LIN {X 0,Y 172.638,Z 369.1,A -85,B 0,C 180,E1 -26067.806,E2 -26067.806} C_VEL
LIN {X 0,Y 170.453,Z 370.698,A -85,B 0,C 180,E1 -26067.724,E2 -26067.724} C_VEL
LIN {X 0,Y 167.759,Z 372.433,A -85,B 0,C 180,E1 -26068.163,E2 -26068.163} C_VEL
LIN {X 0,Y 165.128,Z 374.03,A -85,B 0,C 180,E1 -26069.021,E2 -26069.021} C_VEL
LIN {X 0,Y 159.69,Z 377.088,A -85,B 0,C 180,E1 -26071.335,E2 -26071.335} C_VEL
LIN {X 0,Y 157.543,Z 378.251,A -85,B 0,C 180,E1 -26071.948,E2 -26071.948} C_VEL
LIN {X 0,Y 147.13,Z 383.164,A -85,B 0,C 180,E1 -26074.539,E2 -26074.539} C_VEL
LIN {X 0,Y 136.791,Z 386.889,A -85,B 0,C 180,E1 -26077.644,E2 -26077.644} C_VEL
LIN {X 0,Y 125.587,Z 389.614,A -85,B 0,C 180,E1 -26082.061,E2 -26082.061} C_VEL
LIN {X 0,Y 115.177,Z 390.768,A -85,B 0,C 180,E1 -26087.515,E2 -26087.515} C_VEL
LIN {X 0,Y 105.941,Z 390.198,A -85,B 0,C 180,E1 -26094.344,E2 -26094.344} C_VEL
LIN {X 0,Y 100.509,Z 388.699,A -85,B 0,C 180,E1 -26100.001,E2 -26100.001} C_VEL
LIN {X 0,Y 97.504,Z 387.177,A -85,B 0,C 180,E1 -26104.134,E2 -26104.134} C_VEL
LIN {X 0,Y 93.505,Z 383.221,A -85,B 0,C 180,E1 -26112.269,E2 -26112.269} C_VEL
LIN {X 0,Y 91.521,Z 378.192,A -85,B 0,C 180,E1 -26120.181,E2 -26120.181} C_VEL
LIN {X 0,Y 91.194,Z 372.228,A -85,B 0,C 180,E1 -26127.543,E2 -26127.543} C_VEL
LIN {X 0,Y 91.607,Z 365.87,A -85,B 0,C 180,E1 -26133.796,E2 -26133.796} C_VEL
LIN {X 0,Y 92.588,Z 357.724,A -85,B 0,C 180,E1 -26140.216,E2 -26140.216} C_VEL
LIN {X 0,Y 94.126,Z 348.531,A -85,B 0,C 180,E1 -26145.946,E2 -26145.946} C_VEL
LIN {X 0,Y 96.068,Z 338.761,A -85,B 0,C 180,E1 -26150.765,E2 -26150.765} C_VEL
LIN {X 0,Y 98.32,Z 327.543,A -85,B 0,C 180,E1 -26155.117,E2 -26155.117} C_VEL
LIN {X 0,Y 100.753,Z 315.315,A -85,B 0,C 180,E1 -26158.707,E2 -26158.707} C_VEL
LIN {X 0,Y 102.943,Z 302.841,A -85,B 0,C 180,E1 -26161.448,E2 -26161.448} C_VEL
LIN {X 0,Y 104.614,Z 289.402,A -85,B 0,C 180,E1 -26163.561,E2 -26163.561} C_VEL
LIN {X 0,Y 106.685,Z 268.345,A -85,B 0,C 180,E1 -26165.639,E2 -26165.639} C_VEL
LIN {X 0,Y 109.722,Z 233.038,A -85,B 0,C 180,E1 -26168.778,E2 -26168.778} C_VEL
LIN {X 0,Y 103.431,Z 215.21,A -85,B 0,C 180,E1 -26172.045,E2 -26172.045} C_VEL
LIN {X 0,Y 97.31,Z 199.967,A -85,B 0,C 180,E1 -26175.421,E2 -26175.421} C_VEL
LIN {X 0,Y 94.113,Z 192.132,A -85,B 0,C 180,E1 -26177.325,E2 -26177.325} C_VEL
LIN {X 0,Y 94.078,Z 191.767,A -85,B 0,C 180,E1 -26177.594,E2 -26177.594} C_VEL
LIN {X 0,Y 94.163,Z 191.756,A -85,B 0,C 180,E1 -26181.411,E2 -26181.411} C_VEL
LIN {X 0,Y 94.758,Z 191.674,A -85,B 0,C 180,E1 -26189.996,E2 -26189.996} C_VEL
LIN {X 0,Y 94.134,Z 191.751,A -85,B 0,C 180,E1 -26198.584,E2 -26198.584} C_VEL
LIN {X 0,Y 93.959,Z 191.781,A -85,B 0,C 180,E1 -26203.492,E2 -26203.492} C_VEL
LIN {X 0,Y 93.642,Z 191.82,A -85,B 0,C 180,E1 -26212.036,E2 -26212.036} C_VEL
LIN {X 0,Y 93.586,Z 191.823,A -85,B 0,C 180,E1 -26216.777,E2 -26216.777} C_VEL
LIN {X 0,Y 93.58,Z 191.822,A -85,B 0,C 180,E1 -26224.296,E2 -26224.296} C_VEL
LIN {X 0,Y 93.524,Z 191.827,A -85,B 0,C 180,E1 -26232.551,E2 -26232.551} C_VEL
LIN {X 0,Y 93.527,Z 191.83,A -85,B 0,C 180,E1 -26238.71,E2 -26238.71} C_VEL
LIN {X 0,Y 93.579,Z 191.827,A -85,B 0,C 180,E1 -26245.695,E2 -26245.695} C_VEL
LIN {X 0,Y 93.637,Z 191.82,A -85,B 0,C 180,E1 -26254.237,E2 -26254.237} C_VEL
LIN {X 0,Y 93.646,Z 191.813,A -85,B 0,C 180,E1 -26257.96,E2 -26257.96} C_VEL
LIN {X 0,Y 94.009,Z 191.771,A -85,B 0,C 180,E1 -26267.039,E2 -26267.039} C_VEL
LIN {X 0,Y 94.152,Z 191.756,A -85,B 0,C 180,E1 -26271.413,E2 -26271.413} C_VEL
LIN {X 0,Y 94.749,Z 191.68,A -85,B 0,C 180,E1 -26279.999,E2 -26279.999} C_VEL
LIN {X 0,Y 94.125,Z 191.758,A -85,B 0,C 180,E1 -26288.587,E2 -26288.587} C_VEL
LIN {X 0,Y 93.951,Z 191.781,A -85,B 0,C 180,E1 -26293.494,E2 -26293.494} C_VEL
LIN {X 0,Y 93.636,Z 191.821,A -85,B 0,C 180,E1 -26302.041,E2 -26302.041} C_VEL
LIN {X 0,Y 93.58,Z 191.822,A -85,B 0,C 180,E1 -26306.782,E2 -26306.782} C_VEL
LIN {X 0,Y 93.576,Z 191.825,A -85,B 0,C 180,E1 -26314.301,E2 -26314.301} C_VEL
LIN {X 0,Y 93.585,Z 191.828,A -85,B 0,C 180,E1 -26319.821,E2 -26319.821} C_VEL
LIN {X 0,Y 94.705,Z 194.871,A -85,B 0,C 180,E1 -26320.588,E2 -26320.588} C_VEL
LIN {X 0,Y 101.84,Z 211.018,A -85,B 0,C 180,E1 -26324.497,E2 -26324.497} C_VEL
LIN {X 0,Y 108.216,Z 233.918,A -85,B 0,C 180,E1 -26328.406,E2 -26328.406} C_VEL
LIN {X 0,Y 108.775,Z 238.103,A -85,B 0,C 180,E1 -26328.95,E2 -26328.95} C_VEL
LIN {X 0,Y 109.169,Z 245.942,A -85,B 0,C 180,E1 -26329.835,E2 -26329.835} C_VEL
LIN {X 0,Y 105.151,Z 291.907,A -85,B 0,C 180,E1 -26334.066,E2 -26334.066} C_VEL
LIN {X 0,Y 103.46,Z 304.913,A -85,B 0,C 180,E1 -26335.92,E2 -26335.92} C_VEL
LIN {X 0,Y 101.232,Z 318.223,A -85,B 0,C 180,E1 -26338.626,E2 -26338.626} C_VEL
LIN {X 0,Y 98.938,Z 330.029,A -85,B 0,C 180,E1 -26341.931,E2 -26341.931} C_VEL
LIN {X 0,Y 96.46,Z 342.113,A -85,B 0,C 180,E1 -26346.38,E2 -26346.38} C_VEL
LIN {X 0,Y 94.41,Z 352.803,A -85,B 0,C 180,E1 -26351.56,E2 -26351.56} C_VEL
LIN {X 0,Y 93.041,Z 361.54,A -85,B 0,C 180,E1 -26356.906,E2 -26356.906} C_VEL
LIN {X 0,Y 92.355,Z 368.876,A -85,B 0,C 180,E1 -26362.495,E2 -26362.495} C_VEL
LIN {X 0,Y 92.285,Z 375.689,A -85,B 0,C 180,E1 -26368.913,E2 -26368.913} C_VEL
LIN {X 0,Y 92.355,Z 378.572,A -85,B 0,C 180,E1 -26372.184,E2 -26372.184} C_VEL
LIN {X 0,Y 92.189,Z 383.199,A -85,B 0,C 180,E1 -26378.774,E2 -26378.774} C_VEL
LIN {X 0,Y 93.115,Z 386.821,A -85,B 0,C 180,E1 -26385.321,E2 -26385.321} C_VEL
LIN {X 0,Y 95.224,Z 389.563,A -85,B 0,C 180,E1 -26391.659,E2 -26391.659} C_VEL
LIN {X 0,Y 99.89,Z 392.01,A -85,B 0,C 180,E1 -26399.509,E2 -26399.509} C_VEL
LIN {X 0,Y 106.598,Z 393.144,A -85,B 0,C 180,E1 -26406.4,E2 -26406.4} C_VEL
LIN {X 0,Y 114.858,Z 392.97,A -85,B 0,C 180,E1 -26412.309,E2 -26412.309} C_VEL
LIN {X 0,Y 124.234,Z 391.453,A -85,B 0,C 180,E1 -26417.346,E2 -26417.346} C_VEL
LIN {X 0,Y 134.749,Z 388.583,A -85,B 0,C 180,E1 -26421.479,E2 -26421.479} C_VEL
LIN {X 0,Y 146.079,Z 384.264,A -85,B 0,C 180,E1 -26424.878,E2 -26424.878} C_VEL
LIN {X 0,Y 154.429,Z 380.236,A -85,B 0,C 180,E1 -26426.9,E2 -26426.9} C_VEL
LIN {X 0,Y 164.165,Z 374.602,A -85,B 0,C 180,E1 -26428.898,E2 -26428.898} C_VEL
LIN {X 0,Y 166.024,Z 373.418,A -85,B 0,C 180,E1 -26429.237,E2 -26429.237} C_VEL
LIN {X 0,Y 167.851,Z 372.157,A -85,B 0,C 180,E1 -26429.839,E2 -26429.839} C_VEL
LIN {X 0,Y 157.543,Z 378.251,A -85,B 0,C 180,E1 -26431.948,E2 -26431.948} C_VEL
LIN {X 0,Y 152.658,Z 380.71,A -85,B 0,C 180,E1 -26432.791,E2 -26432.791} C_VEL
LIN {X 0,Y 140.141,Z 385.717,A -85,B 0,C 180,E1 -26434.113,E2 -26434.113} C_VEL
LIN {X 0,Y 134.791,Z 387.382,A -85,B 0,C 180,E1 -26434.902,E2 -26434.902} C_VEL
LIN {X 0,Y 129.86,Z 388.621,A -85,B 0,C 180,E1 -26436.166,E2 -26436.166} C_VEL
LIN {X 0,Y 119.503,Z 390.467,A -85,B 0,C 180,E1 -26440.222,E2 -26440.222} C_VEL
LIN {X 0,Y 108.749,Z 391.045,A -85,B 0,C 180,E1 -26445.799,E2 -26445.799} C_VEL
LIN {X 0,Y 100.286,Z 390.123,A -85,B 0,C 180,E1 -26451.944,E2 -26451.944} C_VEL
LIN {X 0,Y 92.745,Z 387.564,A -85,B 0,C 180,E1 -26460.001,E2 -26460.001} C_VEL
LIN {X 0,Y 88.53,Z 384.524,A -85,B 0,C 180,E1 -26466.84,E2 -26466.84} C_VEL
LIN {X 0,Y 85.732,Z 380.425,A -85,B 0,C 180,E1 -26474.238,E2 -26474.238} C_VEL
LIN {X 0,Y 84.452,Z 375.617,A -85,B 0,C 180,E1 -26481.4,E2 -26481.4} C_VEL
LIN {X 0,Y 84.254,Z 369.652,A -85,B 0,C 180,E1 -26488.663,E2 -26488.663} C_VEL
LIN {X 0,Y 84.83,Z 362.659,A -85,B 0,C 180,E1 -26495.448,E2 -26495.448} C_VEL
LIN {X 0,Y 86.008,Z 353.907,A -85,B 0,C 180,E1 -26502.219,E2 -26502.219} C_VEL
LIN {X 0,Y 87.916,Z 343.463,A -85,B 0,C 180,E1 -26508.52,E2 -26508.52} C_VEL
LIN {X 0,Y 89.928,Z 333.534,A -85,B 0,C 180,E1 -26513.232,E2 -26513.232} C_VEL
LIN {X 0,Y 92.4,Z 322.052,A -85,B 0,C 180,E1 -26517.472,E2 -26517.472} C_VEL
LIN {X 0,Y 94.926,Z 309.313,A -85,B 0,C 180,E1 -26520.983,E2 -26520.983} C_VEL
LIN {X 0,Y 96.998,Z 296.051,A -85,B 0,C 180,E1 -26523.619,E2 -26523.619} C_VEL
LIN {X 0,Y 98.656,Z 281.536,A -85,B 0,C 180,E1 -26525.543,E2 -26525.543} C_VEL
LIN {X 0,Y 103.049,Z 234.956,A -85,B 0,C 180,E1 -26529.929,E2 -26529.929} C_VEL
LIN {X 0,Y 98.97,Z 222.631,A -85,B 0,C 180,E1 -26532.297,E2 -26532.297} C_VEL
LIN {X 0,Y 92.348,Z 205.494,A -85,B 0,C 180,E1 -26536.157,E2 -26536.157} C_VEL
LIN {X 0,Y 87.771,Z 195.022,A -85,B 0,C 180,E1 -26539.047,E2 -26539.047} C_VEL
LIN {X 0,Y 87.046,Z 192.643,A -85,B 0,C 180,E1 -26539.83,E2 -26539.83} C_VEL
LIN {X 0,Y 87.688,Z 192.555,A -85,B 0,C 180,E1 -26549.996,E2 -26549.996} C_VEL
LIN {X 0,Y 87.027,Z 192.638,A -85,B 0,C 180,E1 -26559.291,E2 -26559.291} C_VEL
LIN {X 0,Y 86.86,Z 192.664,A -85,B 0,C 180,E1 -26564.044,E2 -26564.044} C_VEL
LIN {X 0,Y 86.593,Z 192.696,A -85,B 0,C 180,E1 -26568.94,E2 -26568.94} C_VEL
LIN {X 0,Y 86.554,Z 192.699,A -85,B 0,C 180,E1 -26576.722,E2 -26576.722} C_VEL
LIN {X 0,Y 86.499,Z 192.708,A -85,B 0,C 180,E1 -26585.657,E2 -26585.657} C_VEL
LIN {X 0,Y 86.468,Z 192.707,A -85,B 0,C 180,E1 -26592.985,E2 -26592.985} C_VEL
LIN {X 0,Y 86.449,Z 192.71,A -85,B 0,C 180,E1 -26599.429,E2 -26599.429} C_VEL
LIN {X 0,Y 86.523,Z 192.707,A -85,B 0,C 180,E1 -26605.346,E2 -26605.346} C_VEL
LIN {X 0,Y 86.559,Z 192.703,A -85,B 0,C 180,E1 -26613.259,E2 -26613.259} C_VEL
LIN {X 0,Y 86.592,Z 192.699,A -85,B 0,C 180,E1 -26621.054,E2 -26621.054} C_VEL
LIN {X 0,Y 86.856,Z 192.658,A -85,B 0,C 180,E1 -26626.148,E2 -26626.148} C_VEL
LIN {X 0,Y 87.055,Z 192.64,A -85,B 0,C 180,E1 -26630.707,E2 -26630.707} C_VEL
LIN {X 0,Y 87.678,Z 192.561,A -85,B 0,C 180,E1 -26639.999,E2 -26639.999} C_VEL
LIN {X 0,Y 87.019,Z 192.64,A -85,B 0,C 180,E1 -26649.295,E2 -26649.295} C_VEL
LIN {X 0,Y 86.853,Z 192.667,A -85,B 0,C 180,E1 -26654.048,E2 -26654.048} C_VEL
LIN {X 0,Y 86.585,Z 192.692,A -85,B 0,C 180,E1 -26658.945,E2 -26658.945} C_VEL
LIN {X 0,Y 86.548,Z 192.697,A -85,B 0,C 180,E1 -26666.727,E2 -26666.727} C_VEL
LIN {X 0,Y 86.471,Z 192.704,A -85,B 0,C 180,E1 -26675.641,E2 -26675.641} C_VEL
LIN {X 0,Y 86.51,Z 192.893,A -85,B 0,C 180,E1 -26677.575,E2 -26677.575} C_VEL
LIN {X 0,Y 87.529,Z 195.553,A -85,B 0,C 180,E1 -26678.319,E2 -26678.319} C_VEL
LIN {X 0,Y 92.221,Z 205.62,A -85,B 0,C 180,E1 -26681.194,E2 -26681.194} C_VEL
LIN {X 0,Y 96.159,Z 215.384,A -85,B 0,C 180,E1 -26683.52,E2 -26683.52} C_VEL
LIN {X 0,Y 102.028,Z 237.053,A -85,B 0,C 180,E1 -26687.476,E2 -26687.476} C_VEL
LIN {X 0,Y 102.435,Z 246.588,A -85,B 0,C 180,E1 -26688.628,E2 -26688.628} C_VEL
LIN {X 0,Y 98.298,Z 291.946,A -85,B 0,C 180,E1 -26693.062,E2 -26693.062} C_VEL
LIN {X 0,Y 96.341,Z 306.14,A -85,B 0,C 180,E1 -26695.26,E2 -26695.26} C_VEL
LIN {X 0,Y 94.222,Z 318.099,A -85,B 0,C 180,E1 -26697.901,E2 -26697.901} C_VEL
LIN {X 0,Y 91.871,Z 329.891,A -85,B 0,C 180,E1 -26701.442,E2 -26701.442} C_VEL
LIN {X 0,Y 89.325,Z 341.868,A -85,B 0,C 180,E1 -26706.224,E2 -26706.224} C_VEL
LIN {X 0,Y 87.44,Z 351.526,A -85,B 0,C 180,E1 -26711.25,E2 -26711.25} C_VEL
LIN {X 0,Y 86.054,Z 360.36,A -85,B 0,C 180,E1 -26717.027,E2 -26717.027} C_VEL
LIN {X 0,Y 85.397,Z 367.554,A -85,B 0,C 180,E1 -26722.814,E2 -26722.814} C_VEL
LIN {X 0,Y 85.354,Z 373.709,A -85,B 0,C 180,E1 -26728.825,E2 -26728.825} C_VEL
LIN {X 0,Y 85.445,Z 376.765,A -85,B 0,C 180,E1 -26732.361,E2 -26732.361} C_VEL
LIN {X 0,Y 85.35,Z 381.668,A -85,B 0,C 180,E1 -26739.483,E2 -26739.483} C_VEL
LIN {X 0,Y 87.053,Z 386.605,A -85,B 0,C 180,E1 -26748.844,E2 -26748.844} C_VEL
LIN {X 0,Y 90.932,Z 390.065,A -85,B 0,C 180,E1 -26757.632,E2 -26757.632} C_VEL
LIN {X 0,Y 97.206,Z 392.165,A -85,B 0,C 180,E1 -26765.342,E2 -26765.342} C_VEL
LIN {X 0,Y 105.243,Z 392.954,A -85,B 0,C 180,E1 -26771.901,E2 -26771.901} C_VEL
LIN {X 0,Y 114.484,Z 392.455,A -85,B 0,C 180,E1 -26777.452,E2 -26777.452} C_VEL
LIN {X 0,Y 124.898,Z 390.666,A -85,B 0,C 180,E1 -26781.983,E2 -26781.983} C_VEL
LIN {X 0,Y 136.239,Z 387.523,A -85,B 0,C 180,E1 -26785.631,E2 -26785.631} C_VEL
LIN {X 0,Y 148.218,Z 382.837,A -85,B 0,C 180,E1 -26788.598,E2 -26788.598} C_VEL
LIN {X 0,Y 153.766,Z 380.197,A -85,B 0,C 180,E1 -26789.817,E2 -26789.817} C_VEL
LIN {X 0,Y 142.772,Z 384.797,A -85,B 0,C 180,E1 -26792.386,E2 -26792.386} C_VEL
LIN {X 0,Y 129.86,Z 388.621,A -85,B 0,C 180,E1 -26796.166,E2 -26796.166} C_VEL
LIN {X 0,Y 124.946,Z 389.646,A -85,B 0,C 180,E1 -26797.576,E2 -26797.576} C_VEL
LIN {X 0,Y 115.956,Z 390.886,A -85,B 0,C 180,E1 -26799.48,E2 -26799.48} C_VEL
LIN {X 0,Y 107.125,Z 391.284,A -85,B 0,C 180,E1 -26801.743,E2 -26801.743} C_VEL
LIN {X 0,Y 102.58,Z 391.108,A -85,B 0,C 180,E1 -26803.784,E2 -26803.784} C_VEL
LIN {X 0,Y 97.135,Z 390.428,A -85,B 0,C 180,E1 -26807.465,E2 -26807.465} C_VEL
LIN {X 0,Y 92.411,Z 389.334,A -85,B 0,C 180,E1 -26811.389,E2 -26811.389} C_VEL
LIN {X 0,Y 84.94,Z 386.05,A -85,B 0,C 180,E1 -26820.001,E2 -26820.001} C_VEL
LIN {X 0,Y 80.873,Z 382.427,A -85,B 0,C 180,E1 -26827.491,E2 -26827.491} C_VEL
LIN {X 0,Y 78.306,Z 377.701,A -85,B 0,C 180,E1 -26835.621,E2 -26835.621} C_VEL
LIN {X 0,Y 77.29,Z 371.334,A -85,B 0,C 180,E1 -26844.581,E2 -26844.581} C_VEL
LIN {X 0,Y 77.469,Z 365.374,A -85,B 0,C 180,E1 -26851.444,E2 -26851.444} C_VEL
LIN {X 0,Y 78.36,Z 357.328,A -85,B 0,C 180,E1 -26858.891,E2 -26858.891} C_VEL
LIN {X 0,Y 80.032,Z 347.091,A -85,B 0,C 180,E1 -26866.243,E2 -26866.243} C_VEL
LIN {X 0,Y 82.236,Z 336.455,A -85,B 0,C 180,E1 -26872.151,E2 -26872.151} C_VEL
LIN {X 0,Y 84.715,Z 324.699,A -85,B 0,C 180,E1 -26877.14,E2 -26877.14} C_VEL
LIN {X 0,Y 87.377,Z 312.075,A -85,B 0,C 180,E1 -26881.141,E2 -26881.141} C_VEL
LIN {X 0,Y 89.769,Z 298.591,A -85,B 0,C 180,E1 -26884.205,E2 -26884.205} C_VEL
LIN {X 0,Y 91.489,Z 285.046,A -85,B 0,C 180,E1 -26886.325,E2 -26886.325} C_VEL
LIN {X 0,Y 96.269,Z 235.616,A -85,B 0,C 180,E1 -26891.403,E2 -26891.403} C_VEL
LIN {X 0,Y 89.652,Z 216.903,A -85,B 0,C 180,E1 -26895.484,E2 -26895.484} C_VEL
LIN {X 0,Y 82.617,Z 199.461,A -85,B 0,C 180,E1 -26900.355,E2 -26900.355} C_VEL
LIN {X 0,Y 80.163,Z 194.324,A -85,B 0,C 180,E1 -26902.122,E2 -26902.122} C_VEL
LIN {X 0,Y 80.019,Z 193.518,A -85,B 0,C 180,E1 -26902.425,E2 -26902.425} C_VEL
LIN {X 0,Y 80.618,Z 193.435,A -85,B 0,C 180,E1 -26909.996,E2 -26909.996} C_VEL
LIN {X 0,Y 79.912,Z 193.526,A -85,B 0,C 180,E1 -26920.126,E2 -26920.126} C_VEL
LIN {X 0,Y 79.687,Z 193.553,A -85,B 0,C 180,E1 -26925.338,E2 -26925.338} C_VEL
LIN {X 0,Y 79.47,Z 193.586,A -85,B 0,C 180,E1 -26930.712,E2 -26930.712} C_VEL
LIN {X 0,Y 79.457,Z 193.586,A -85,B 0,C 180,E1 -26937.806,E2 -26937.806} C_VEL
LIN {X 0,Y 79.365,Z 193.594,A -85,B 0,C 180,E1 -26942.089,E2 -26942.089} C_VEL
LIN {X 0,Y 79.359,Z 193.6,A -85,B 0,C 180,E1 -26948.304,E2 -26948.304} C_VEL
LIN {X 0,Y 79.381,Z 193.597,A -85,B 0,C 180,E1 -26955.089,E2 -26955.089} C_VEL
LIN {X 0,Y 79.379,Z 193.595,A -85,B 0,C 180,E1 -26962.822,E2 -26962.822} C_VEL
LIN {X 0,Y 79.365,Z 193.592,A -85,B 0,C 180,E1 -26967.904,E2 -26967.904} C_VEL
LIN {X 0,Y 79.5,Z 193.582,A -85,B 0,C 180,E1 -26973.766,E2 -26973.766} C_VEL
LIN {X 0,Y 79.47,Z 193.584,A -85,B 0,C 180,E1 -26979.282,E2 -26979.282} C_VEL
LIN {X 0,Y 79.781,Z 193.539,A -85,B 0,C 180,E1 -26985.679,E2 -26985.679} C_VEL
LIN {X 0,Y 79.93,Z 193.529,A -85,B 0,C 180,E1 -26989.87,E2 -26989.87} C_VEL
LIN {X 0,Y 80.608,Z 193.441,A -85,B 0,C 180,E1 -26999.999,E2 -26999.999} C_VEL
LIN {X 0,Y 79.903,Z 193.524,A -85,B 0,C 180,E1 -27010.131,E2 -27010.131} C_VEL
LIN {X 0,Y 79.679,Z 193.56,A -85,B 0,C 180,E1 -27015.343,E2 -27015.343} C_VEL
LIN {X 0,Y 79.463,Z 193.583,A -85,B 0,C 180,E1 -27020.717,E2 -27020.717} C_VEL
LIN {X 0,Y 79.436,Z 193.582,A -85,B 0,C 180,E1 -27027.791,E2 -27027.791} C_VEL
LIN {X 0,Y 79.489,Z 193.673,A -85,B 0,C 180,E1 -27034.884,E2 -27034.884} C_VEL
LIN {X 0,Y 80.538,Z 196.605,A -85,B 0,C 180,E1 -27035.788,E2 -27035.788} C_VEL
LIN {X 0,Y 84.871,Z 205.502,A -85,B 0,C 180,E1 -27038.772,E2 -27038.772} C_VEL
LIN {X 0,Y 89.859,Z 217.528,A -85,B 0,C 180,E1 -27042.042,E2 -27042.042} C_VEL
LIN {X 0,Y 95.399,Z 238.371,A -85,B 0,C 180,E1 -27046.101,E2 -27046.101} C_VEL
LIN {X 0,Y 95.728,Z 247.096,A -85,B 0,C 180,E1 -27047.235,E2 -27047.235} C_VEL
LIN {X 0,Y 91.485,Z 291.748,A -85,B 0,C 180,E1 -27051.91,E2 -27051.91} C_VEL
LIN {X 0,Y 89.44,Z 305.785,A -85,B 0,C 180,E1 -27054.243,E2 -27054.243} C_VEL
LIN {X 0,Y 87.257,Z 317.687,A -85,B 0,C 180,E1 -27057.071,E2 -27057.071} C_VEL
LIN {X 0,Y 84.848,Z 329.439,A -85,B 0,C 180,E1 -27060.885,E2 -27060.885} C_VEL
LIN {X 0,Y 82.212,Z 341.413,A -85,B 0,C 180,E1 -27066.047,E2 -27066.047} C_VEL
LIN {X 0,Y 80.156,Z 352.071,A -85,B 0,C 180,E1 -27072.133,E2 -27072.133} C_VEL
LIN {X 0,Y 78.748,Z 362.348,A -85,B 0,C 180,E1 -27079.722,E2 -27079.722} C_VEL
LIN {X 0,Y 78.425,Z 370.456,A -85,B 0,C 180,E1 -27087.436,E2 -27087.436} C_VEL
LIN {X 0,Y 78.579,Z 374.833,A -85,B 0,C 180,E1 -27092.567,E2 -27092.567} C_VEL
LIN {X 0,Y 78.575,Z 379.992,A -85,B 0,C 180,E1 -27100.309,E2 -27100.309} C_VEL
LIN {X 0,Y 80.457,Z 385.32,A -85,B 0,C 180,E1 -27110.455,E2 -27110.455} C_VEL
LIN {X 0,Y 84.768,Z 389.029,A -85,B 0,C 180,E1 -27119.836,E2 -27119.836} C_VEL
LIN {X 0,Y 91.52,Z 391.464,A -85,B 0,C 180,E1 -27127.908,E2 -27127.908} C_VEL
LIN {X 0,Y 100.08,Z 392.606,A -85,B 0,C 180,E1 -27134.611,E2 -27134.611} C_VEL
LIN {X 0,Y 110.392,Z 392.434,A -85,B 0,C 180,E1 -27140.459,E2 -27140.459} C_VEL
LIN {X 0,Y 120.672,Z 391.061,A -85,B 0,C 180,E1 -27144.629,E2 -27144.629} C_VEL
LIN {X 0,Y 132.389,Z 388.294,A -85,B 0,C 180,E1 -27148.148,E2 -27148.148} C_VEL
LIN {X 0,Y 138.472,Z 386.374,A -85,B 0,C 180,E1 -27149.639,E2 -27149.639} C_VEL
LIN {X 0,Y 137.457,Z 386.659,A -85,B 0,C 180,E1 -27150.369,E2 -27150.369} C_VEL
LIN {X 0,Y 125.413,Z 389.626,A -85,B 0,C 180,E1 -27153.723,E2 -27153.723} C_VEL
LIN {X 0,Y 113.507,Z 391.115,A -85,B 0,C 180,E1 -27158.192,E2 -27158.192} C_VEL
LIN {X 0,Y 102.58,Z 391.108,A -85,B 0,C 180,E1 -27163.784,E2 -27163.784} C_VEL
LIN {X 0,Y 98.197,Z 390.736,A -85,B 0,C 180,E1 -27166.042,E2 -27166.042} C_VEL
LIN {X 0,Y 90.163,Z 389.329,A -85,B 0,C 180,E1 -27169.487,E2 -27169.487} C_VEL
LIN {X 0,Y 82.682,Z 387.199,A -85,B 0,C 180,E1 -27173.565,E2 -27173.565} C_VEL
LIN {X 0,Y 79.333,Z 385.598,A -85,B 0,C 180,E1 -27176.827,E2 -27176.827} C_VEL
LIN {X 0,Y 74.434,Z 381.416,A -85,B 0,C 180,E1 -27185.419,E2 -27185.419} C_VEL
LIN {X 0,Y 71.504,Z 376.262,A -85,B 0,C 180,E1 -27194.489,E2 -27194.489} C_VEL
LIN {X 0,Y 70.419,Z 370.145,A -85,B 0,C 180,E1 -27203.53,E2 -27203.53} C_VEL
LIN {X 0,Y 70.578,Z 363.513,A -85,B 0,C 180,E1 -27211.521,E2 -27211.521} C_VEL
LIN {X 0,Y 71.329,Z 356.478,A -85,B 0,C 180,E1 -27218.432,E2 -27218.432} C_VEL
LIN {X 0,Y 72.883,Z 346.746,A -85,B 0,C 180,E1 -27226.09,E2 -27226.09} C_VEL
LIN {X 0,Y 75.184,Z 335.972,A -85,B 0,C 180,E1 -27232.616,E2 -27232.616} C_VEL
LIN {X 0,Y 77.869,Z 323.707,A -85,B 0,C 180,E1 -27238.193,E2 -27238.193} C_VEL
LIN {X 0,Y 80.349,Z 312.264,A -85,B 0,C 180,E1 -27242.046,E2 -27242.046} C_VEL
LIN {X 0,Y 82.686,Z 299.665,A -85,B 0,C 180,E1 -27245.156,E2 -27245.156} C_VEL
LIN {X 0,Y 84.525,Z 286.273,A -85,B 0,C 180,E1 -27247.479,E2 -27247.479} C_VEL
LIN {X 0,Y 89.596,Z 236.968,A -85,B 0,C 180,E1 -27252.868,E2 -27252.868} C_VEL
LIN {X 0,Y 82.373,Z 216.473,A -85,B 0,C 180,E1 -27257.942,E2 -27257.942} C_VEL
LIN {X 0,Y 76.009,Z 200.994,A -85,B 0,C 180,E1 -27262.856,E2 -27262.856} C_VEL
LIN {X 0,Y 73.287,Z 195.445,A -85,B 0,C 180,E1 -27265.096,E2 -27265.096} C_VEL
LIN {X 0,Y 73.09,Z 194.381,A -85,B 0,C 180,E1 -27265.514,E2 -27265.514} C_VEL
LIN {X 0,Y 73.545,Z 194.316,A -85,B 0,C 180,E1 -27269.995,E2 -27269.995} C_VEL
LIN {X 0,Y 72.811,Z 194.414,A -85,B 0,C 180,E1 -27281.126,E2 -27281.126} C_VEL
LIN {X 0,Y 72.503,Z 194.445,A -85,B 0,C 180,E1 -27286.901,E2 -27286.901} C_VEL
LIN {X 0,Y 72.36,Z 194.469,A -85,B 0,C 180,E1 -27292.856,E2 -27292.856} C_VEL
LIN {X 0,Y 72.356,Z 194.472,A -85,B 0,C 180,E1 -27299.05,E2 -27299.05} C_VEL
LIN {X 0,Y 72.287,Z 194.477,A -85,B 0,C 180,E1 -27305.68,E2 -27305.68} C_VEL
LIN {X 0,Y 72.241,Z 194.479,A -85,B 0,C 180,E1 -27312.915,E2 -27312.915} C_VEL
LIN {X 0,Y 72.287,Z 194.473,A -85,B 0,C 180,E1 -27321.05,E2 -27321.05} C_VEL
LIN {X 0,Y 72.286,Z 194.481,A -85,B 0,C 180,E1 -27324.312,E2 -27324.312} C_VEL
LIN {X 0,Y 72.353,Z 194.469,A -85,B 0,C 180,E1 -27330.942,E2 -27330.942} C_VEL
LIN {X 0,Y 72.361,Z 194.463,A -85,B 0,C 180,E1 -27337.138,E2 -27337.138} C_VEL
LIN {X 0,Y 72.672,Z 194.424,A -85,B 0,C 180,E1 -27345.239,E2 -27345.239} C_VEL
LIN {X 0,Y 72.821,Z 194.414,A -85,B 0,C 180,E1 -27348.869,E2 -27348.869} C_VEL
LIN {X 0,Y 73.535,Z 194.322,A -85,B 0,C 180,E1 -27359.999,E2 -27359.999} C_VEL
LIN {X 0,Y 72.803,Z 194.408,A -85,B 0,C 180,E1 -27371.131,E2 -27371.131} C_VEL
LIN {X 0,Y 72.496,Z 194.451,A -85,B 0,C 180,E1 -27376.906,E2 -27376.906} C_VEL
LIN {X 0,Y 72.353,Z 194.472,A -85,B 0,C 180,E1 -27382.862,E2 -27382.862} C_VEL
LIN {X 0,Y 72.305,Z 194.479,A -85,B 0,C 180,E1 -27391.495,E2 -27391.495} C_VEL
LIN {X 0,Y 73.468,Z 197.528,A -85,B 0,C 180,E1 -27392.756,E2 -27392.756} C_VEL
LIN {X 0,Y 74.424,Z 199.131,A -85,B 0,C 180,E1 -27393.492,E2 -27393.492} C_VEL
LIN {X 0,Y 79.302,Z 209.305,A -85,B 0,C 180,E1 -27397.228,E2 -27397.228} C_VEL
LIN {X 0,Y 83.907,Z 221.015,A -85,B 0,C 180,E1 -27400.648,E2 -27400.648} C_VEL
LIN {X 0,Y 88.851,Z 239.915,A -85,B 0,C 180,E1 -27404.696,E2 -27404.696} C_VEL
LIN {X 0,Y 89.097,Z 246.934,A -85,B 0,C 180,E1 -27405.674,E2 -27405.674} C_VEL
LIN {X 0,Y 84.603,Z 291.809,A -85,B 0,C 180,E1 -27410.703,E2 -27410.703} C_VEL
LIN {X 0,Y 82.605,Z 305.148,A -85,B 0,C 180,E1 -27413.073,E2 -27413.073} C_VEL
LIN {X 0,Y 80.322,Z 317.124,A -85,B 0,C 180,E1 -27416.102,E2 -27416.102} C_VEL
LIN {X 0,Y 77.812,Z 328.946,A -85,B 0,C 180,E1 -27420.219,E2 -27420.219} C_VEL
LIN {X 0,Y 75.132,Z 340.977,A -85,B 0,C 180,E1 -27425.848,E2 -27425.848} C_VEL
LIN {X 0,Y 73.202,Z 350.713,A -85,B 0,C 180,E1 -27431.824,E2 -27431.824} C_VEL
LIN {X 0,Y 71.921,Z 359.501,A -85,B 0,C 180,E1 -27438.735,E2 -27438.735} C_VEL
LIN {X 0,Y 71.509,Z 366.77,A -85,B 0,C 180,E1 -27445.778,E2 -27445.778} C_VEL
LIN {X 0,Y 71.729,Z 372.748,A -85,B 0,C 180,E1 -27452.813,E2 -27452.813} C_VEL
LIN {X 0,Y 71.715,Z 376.916,A -85,B 0,C 180,E1 -27459.082,E2 -27459.082} C_VEL
LIN {X 0,Y 73.173,Z 382.596,A -85,B 0,C 180,E1 -27469.648,E2 -27469.648} C_VEL
LIN {X 0,Y 76.061,Z 386.043,A -85,B 0,C 180,E1 -27477.521,E2 -27477.521} C_VEL
LIN {X 0,Y 82.117,Z 389.468,A -85,B 0,C 180,E1 -27486.81,E2 -27486.81} C_VEL
LIN {X 0,Y 90.367,Z 391.58,A -85,B 0,C 180,E1 -27494.428,E2 -27494.428} C_VEL
LIN {X 0,Y 100.13,Z 392.419,A -85,B 0,C 180,E1 -27500.546,E2 -27500.546} C_VEL
LIN {X 0,Y 110.948,Z 392.003,A -85,B 0,C 180,E1 -27505.44,E2 -27505.44} C_VEL
LIN {X 0,Y 122.667,Z 390.321,A -85,B 0,C 180,E1 -27509.254,E2 -27509.254} C_VEL
LIN {X 0,Y 123.924,Z 390.038,A -85,B 0,C 180,E1 -27510.322,E2 -27510.322} C_VEL
LIN {X 0,Y 112.421,Z 391.373,A -85,B 0,C 180,E1 -27514.05,E2 -27514.05} C_VEL
LIN {X 0,Y 106.157,Z 391.564,A -85,B 0,C 180,E1 -27516.596,E2 -27516.596} C_VEL
LIN {X 0,Y 96.236,Z 390.944,A -85,B 0,C 180,E1 -27521.701,E2 -27521.701} C_VEL
LIN {X 0,Y 89.481,Z 389.667,A -85,B 0,C 180,E1 -27526.372,E2 -27526.372} C_VEL
LIN {X 0,Y 80.714,Z 386.425,A -85,B 0,C 180,E1 -27535.006,E2 -27535.006} C_VEL
LIN {X 0,Y 79.333,Z 385.598,A -85,B 0,C 180,E1 -27536.827,E2 -27536.827} C_VEL
LIN {X 0,Y 76.325,Z 383.797,A -85,B 0,C 180,E1 -27540.313,E2 -27540.313} C_VEL
LIN {X 0,Y 70.573,Z 380.043,A -85,B 0,C 180,E1 -27545.879,E2 -27545.879} C_VEL
LIN {X 0,Y 65.667,Z 375.531,A -85,B 0,C 180,E1 -27552.128,E2 -27552.128} C_VEL
LIN {X 0,Y 64.158,Z 372.616,A -85,B 0,C 180,E1 -27556.526,E2 -27556.526} C_VEL
LIN {X 0,Y 63.531,Z 365.962,A -85,B 0,C 180,E1 -27566.265,E2 -27566.265} C_VEL
LIN {X 0,Y 63.977,Z 358.339,A -85,B 0,C 180,E1 -27575.16,E2 -27575.16} C_VEL
LIN {X 0,Y 65.211,Z 349.403,A -85,B 0,C 180,E1 -27583.399,E2 -27583.399} C_VEL
LIN {X 0,Y 67.448,Z 338.375,A -85,B 0,C 180,E1 -27591.297,E2 -27591.297} C_VEL
LIN {X 0,Y 69.933,Z 327.224,A -85,B 0,C 180,E1 -27597.318,E2 -27597.318} C_VEL
LIN {X 0,Y 72.875,Z 314.517,A -85,B 0,C 180,E1 -27602.383,E2 -27602.383} C_VEL
LIN {X 0,Y 75.465,Z 301.672,A -85,B 0,C 180,E1 -27606.045,E2 -27606.045} C_VEL
LIN {X 0,Y 77.473,Z 288.155,A -85,B 0,C 180,E1 -27608.719,E2 -27608.719} C_VEL
LIN {X 0,Y 80.412,Z 261.533,A -85,B 0,C 180,E1 -27611.996,E2 -27611.996} C_VEL
LIN {X 0,Y 82.935,Z 238.42,A -85,B 0,C 180,E1 -27614.577,E2 -27614.577} C_VEL
LIN {X 0,Y 76.458,Z 219.612,A -85,B 0,C 180,E1 -27619.653,E2 -27619.653} C_VEL
LIN {X 0,Y 70.517,Z 204.763,A -85,B 0,C 180,E1 -27624.855,E2 -27624.855} C_VEL
LIN {X 0,Y 66.579,Z 196.515,A -85,B 0,C 180,E1 -27628.67,E2 -27628.67} C_VEL
LIN {X 0,Y 66.364,Z 195.211,A -85,B 0,C 180,E1 -27629.236,E2 -27629.236} C_VEL
LIN {X 0,Y 65.875,Z 195.277,A -85,B 0,C 180,E1 -27636.119,E2 -27636.119} C_VEL
LIN {X 0,Y 65.712,Z 195.3,A -85,B 0,C 180,E1 -27642.346,E2 -27642.346} C_VEL
LIN {X 0,Y 65.333,Z 195.343,A -85,B 0,C 180,E1 -27648.822,E2 -27648.822} C_VEL
LIN {X 0,Y 65.21,Z 195.354,A -85,B 0,C 180,E1 -27655.531,E2 -27655.531} C_VEL
LIN {X 0,Y 65.166,Z 195.36,A -85,B 0,C 180,E1 -27662.625,E2 -27662.625} C_VEL
LIN {X 0,Y 65.176,Z 195.358,A -85,B 0,C 180,E1 -27670.988,E2 -27670.988} C_VEL
LIN {X 0,Y 65.195,Z 195.356,A -85,B 0,C 180,E1 -27679.697,E2 -27679.697} C_VEL
LIN {X 0,Y 65.219,Z 195.353,A -85,B 0,C 180,E1 -27689.539,E2 -27689.539} C_VEL
LIN {X 0,Y 65.211,Z 195.36,A -85,B 0,C 180,E1 -27694.461,E2 -27694.461} C_VEL
LIN {X 0,Y 65.575,Z 195.309,A -85,B 0,C 180,E1 -27704.684,E2 -27704.684} C_VEL
LIN {X 0,Y 65.715,Z 195.296,A -85,B 0,C 180,E1 -27707.648,E2 -27707.648} C_VEL
LIN {X 0,Y 66.433,Z 195.207,A -85,B 0,C 180,E1 -27719.999,E2 -27719.999} C_VEL
LIN {X 0,Y 65.704,Z 195.295,A -85,B 0,C 180,E1 -27732.351,E2 -27732.351} C_VEL
LIN {X 0,Y 65.326,Z 195.339,A -85,B 0,C 180,E1 -27738.828,E2 -27738.828} C_VEL
LIN {X 0,Y 65.209,Z 195.354,A -85,B 0,C 180,E1 -27747.606,E2 -27747.606} C_VEL
LIN {X 0,Y 66.296,Z 198.247,A -85,B 0,C 180,E1 -27748.902,E2 -27748.902} C_VEL
LIN {X 0,Y 67.671,Z 200.54,A -85,B 0,C 180,E1 -27750.19,E2 -27750.19} C_VEL
LIN {X 0,Y 71.907,Z 208.928,A -85,B 0,C 180,E1 -27753.981,E2 -27753.981} C_VEL
LIN {X 0,Y 77.041,Z 221.337,A -85,B 0,C 180,E1 -27758.213,E2 -27758.213} C_VEL
LIN {X 0,Y 80.627,Z 234.475,A -85,B 0,C 180,E1 -27761.498,E2 -27761.498} C_VEL
LIN {X 0,Y 82.371,Z 242.088,A -85,B 0,C 180,E1 -27763.166,E2 -27763.166} C_VEL
LIN {X 0,Y 82.387,Z 248.026,A -85,B 0,C 180,E1 -27764.022,E2 -27764.022} C_VEL
LIN {X 0,Y 77.78,Z 291.9,A -85,B 0,C 180,E1 -27769.293,E2 -27769.293} C_VEL
LIN {X 0,Y 75.58,Z 305.767,A -85,B 0,C 180,E1 -27771.978,E2 -27771.978} C_VEL
LIN {X 0,Y 73.046,Z 318.45,A -85,B 0,C 180,E1 -27775.586,E2 -27775.586} C_VEL
LIN {X 0,Y 70.135,Z 331.286,A -85,B 0,C 180,E1 -27780.763,E2 -27780.763} C_VEL
LIN {X 0,Y 67.573,Z 342.678,A -85,B 0,C 180,E1 -27787.05,E2 -27787.05} C_VEL
LIN {X 0,Y 65.723,Z 352.294,A -85,B 0,C 180,E1 -27794.001,E2 -27794.001} C_VEL
LIN {X 0,Y 64.742,Z 361.612,A -85,B 0,C 180,E1 -27802.559,E2 -27802.559} C_VEL
LIN {X 0,Y 64.826,Z 369.375,A -85,B 0,C 180,E1 -27811.558,E2 -27811.558} C_VEL
LIN {X 0,Y 64.978,Z 372.67,A -85,B 0,C 180,E1 -27816.215,E2 -27816.215} C_VEL
LIN {X 0,Y 65.651,Z 378.483,A -85,B 0,C 180,E1 -27826.596,E2 -27826.596} C_VEL
LIN {X 0,Y 68.731,Z 383.508,A -85,B 0,C 180,E1 -27837.402,E2 -27837.402} C_VEL
LIN {X 0,Y 72.936,Z 386.693,A -85,B 0,C 180,E1 -27845.326,E2 -27845.326} C_VEL
LIN {X 0,Y 80.863,Z 389.766,A -85,B 0,C 180,E1 -27854.057,E2 -27854.057} C_VEL
LIN {X 0,Y 90.541,Z 391.588,A -85,B 0,C 180,E1 -27860.921,E2 -27860.921} C_VEL
LIN {X 0,Y 101.316,Z 392.157,A -85,B 0,C 180,E1 -27866.352,E2 -27866.352} C_VEL
LIN {X 0,Y 108.558,Z 391.918,A -85,B 0,C 180,E1 -27869.059,E2 -27869.059} C_VEL
LIN {X 0,Y 109.98,Z 391.738,A -85,B 0,C 180,E1 -27870.494,E2 -27870.494} C_VEL
LIN {X 0,Y 98.909,Z 391.622,A -85,B 0,C 180,E1 -27874.766,E2 -27874.766} C_VEL
LIN {X 0,Y 90.2,Z 390.57,A -85,B 0,C 180,E1 -27879.236,E2 -27879.236} C_VEL
LIN {X 0,Y 79.187,Z 387.565,A -85,B 0,C 180,E1 -27887.513,E2 -27887.513} C_VEL
LIN {X 0,Y 73.023,Z 384.504,A -85,B 0,C 180,E1 -27894.478,E2 -27894.478} C_VEL
LIN {X 0,Y 68.121,Z 380.363,A -85,B 0,C 180,E1 -27902.958,E2 -27902.958} C_VEL
LIN {X 0,Y 64.857,Z 374.925,A -85,B 0,C 180,E1 -27912.751,E2 -27912.751} C_VEL
LIN {X 0,Y 64.158,Z 372.616,A -85,B 0,C 180,E1 -27916.526,E2 -27916.526} C_VEL
LIN {X 0,Y 63.02,Z 369.535,A -85,B 0,C 180,E1 -27920.924,E2 -27920.924} C_VEL
LIN {X 0,Y 61.304,Z 366.086,A -85,B 0,C 180,E1 -27925.079,E2 -27925.079} C_VEL
LIN {X 0,Y 57.999,Z 358.358,A -85,B 0,C 180,E1 -27933.371,E2 -27933.371} C_VEL
LIN {X 0,Y 57.426,Z 354.198,A -85,B 0,C 180,E1 -27937.68,E2 -27937.68} C_VEL
LIN {X 0,Y 57.53,Z 352.78,A -85,B 0,C 180,E1 -27939.119,E2 -27939.119} C_VEL
LIN {X 0,Y 59.205,Z 342.977,A -85,B 0,C 180,E1 -27947.897,E2 -27947.897} C_VEL
LIN {X 0,Y 61.638,Z 332.157,A -85,B 0,C 180,E1 -27955.236,E2 -27955.236} C_VEL
LIN {X 0,Y 64.723,Z 319.433,A -85,B 0,C 180,E1 -27961.584,E2 -27961.584} C_VEL
LIN {X 0,Y 67.651,Z 306.419,A -85,B 0,C 180,E1 -27966.164,E2 -27966.164} C_VEL
LIN {X 0,Y 70.1,Z 292.699,A -85,B 0,C 180,E1 -27969.52,E2 -27969.52} C_VEL
LIN {X 0,Y 72.268,Z 275.972,A -85,B 0,C 180,E1 -27972.044,E2 -27972.044} C_VEL
LIN {X 0,Y 76.296,Z 239.538,A -85,B 0,C 180,E1 -27976.563,E2 -27976.563} C_VEL
LIN {X 0,Y 69.907,Z 220.807,A -85,B 0,C 180,E1 -27982.271,E2 -27982.271} C_VEL
LIN {X 0,Y 65.177,Z 208.601,A -85,B 0,C 180,E1 -27987.12,E2 -27987.12} C_VEL
LIN {X 0,Y 61.221,Z 200.275,A -85,B 0,C 180,E1 -27991.446,E2 -27991.446} C_VEL
LIN {X 0,Y 59.399,Z 197.771,A -85,B 0,C 180,E1 -27993.386,E2 -27993.386} C_VEL
LIN {X 0,Y 58.925,Z 196.145,A -85,B 0,C 180,E1 -27994.269,E2 -27994.269} C_VEL
LIN {X 0,Y 58.589,Z 196.186,A -85,B 0,C 180,E1 -28003.875,E2 -28003.875} C_VEL
LIN {X 0,Y 58.153,Z 196.242,A -85,B 0,C 180,E1 -28011.251,E2 -28011.251} C_VEL
LIN {X 0,Y 58.122,Z 196.245,A -85,B 0,C 180,E1 -28018.918,E2 -28018.918} C_VEL
LIN {X 0,Y 58.018,Z 196.258,A -85,B 0,C 180,E1 -28027.27,E2 -28027.27} C_VEL
LIN {X 0,Y 58.005,Z 196.26,A -85,B 0,C 180,E1 -28036.624,E2 -28036.624} C_VEL
LIN {X 0,Y 58.017,Z 196.255,A -85,B 0,C 180,E1 -28042.719,E2 -28042.719} C_VEL
LIN {X 0,Y 58.121,Z 196.242,A -85,B 0,C 180,E1 -28051.072,E2 -28051.072} C_VEL
LIN {X 0,Y 58.152,Z 196.235,A -85,B 0,C 180,E1 -28058.74,E2 -28058.74} C_VEL
LIN {X 0,Y 58.587,Z 196.179,A -85,B 0,C 180,E1 -28066.117,E2 -28066.117} C_VEL
LIN {X 0,Y 58.765,Z 196.157,A -85,B 0,C 180,E1 -28073.13,E2 -28073.13} C_VEL
LIN {X 0,Y 59.325,Z 196.092,A -85,B 0,C 180,E1 -28079.998,E2 -28079.998} C_VEL
LIN {X 0,Y 58.753,Z 196.167,A -85,B 0,C 180,E1 -28086.869,E2 -28086.869} C_VEL
LIN {X 0,Y 58.465,Z 196.201,A -85,B 0,C 180,E1 -28095.938,E2 -28095.938} C_VEL
LIN {X 0,Y 58.105,Z 196.247,A -85,B 0,C 180,E1 -28102.441,E2 -28102.441} C_VEL
LIN {X 0,Y 59.149,Z 199.119,A -85,B 0,C 180,E1 -28104.105,E2 -28104.105} C_VEL
LIN {X 0,Y 60.799,Z 201.529,A -85,B 0,C 180,E1 -28105.917,E2 -28105.917} C_VEL
LIN {X 0,Y 65.091,Z 209.648,A -85,B 0,C 180,E1 -28110.443,E2 -28110.443} C_VEL
LIN {X 0,Y 69.556,Z 220.24,A -85,B 0,C 180,E1 -28114.854,E2 -28114.854} C_VEL
LIN {X 0,Y 72.127,Z 227.676,A -85,B 0,C 180,E1 -28117.296,E2 -28117.296} C_VEL
LIN {X 0,Y 75.885,Z 243.342,A -85,B 0,C 180,E1 -28121.256,E2 -28121.256} C_VEL
LIN {X 0,Y 75.799,Z 249.09,A -85,B 0,C 180,E1 -28122.126,E2 -28122.126} C_VEL
LIN {X 0,Y 71.043,Z 291.539,A -85,B 0,C 180,E1 -28127.635,E2 -28127.635} C_VEL
LIN {X 0,Y 68.861,Z 304.682,A -85,B 0,C 180,E1 -28130.373,E2 -28130.373} C_VEL
LIN {X 0,Y 66.203,Z 317.519,A -85,B 0,C 180,E1 -28134.284,E2 -28134.284} C_VEL
LIN {X 0,Y 63.153,Z 330.466,A -85,B 0,C 180,E1 -28139.955,E2 -28139.955} C_VEL
LIN {X 0,Y 60.493,Z 341.978,A -85,B 0,C 180,E1 -28146.921,E2 -28146.921} C_VEL
LIN {X 0,Y 58.649,Z 351.529,A -85,B 0,C 180,E1 -28154.586,E2 -28154.586} C_VEL
LIN {X 0,Y 57.859,Z 359.895,A -85,B 0,C 180,E1 -28163.029,E2 -28163.029} C_VEL
LIN {X 0,Y 58.023,Z 366.881,A -85,B 0,C 180,E1 -28171.741,E2 -28171.741} C_VEL
LIN {X 0,Y 58.277,Z 371.39,A -85,B 0,C 180,E1 -28178.676,E2 -28178.676} C_VEL
LIN {X 0,Y 59.569,Z 377.641,A -85,B 0,C 180,E1 -28190.735,E2 -28190.735} C_VEL
LIN {X 0,Y 64.066,Z 383.114,A -85,B 0,C 180,E1 -28203.27,E2 -28203.27} C_VEL
LIN {X 0,Y 71.392,Z 387.179,A -85,B 0,C 180,E1 -28213.565,E2 -28213.565} C_VEL
LIN {X 0,Y 80.908,Z 389.98,A -85,B 0,C 180,E1 -28221.43,E2 -28221.43} C_VEL
LIN {X 0,Y 91.776,Z 391.54,A -85,B 0,C 180,E1 -28227.396,E2 -28227.396} C_VEL
LIN {X 0,Y 97.567,Z 391.865,A -85,B 0,C 180,E1 -28229.82,E2 -28229.82} C_VEL
LIN {X 0,Y 96.92,Z 391.785,A -85,B 0,C 180,E1 -28230.484,E2 -28230.484} C_VEL
LIN {X 0,Y 84.336,Z 389.957,A -85,B 0,C 180,E1 -28236.453,E2 -28236.453} C_VEL
LIN {X 0,Y 74.434,Z 387.036,A -85,B 0,C 180,E1 -28243.546,E2 -28243.546} C_VEL
LIN {X 0,Y 67.429,Z 383.542,A -85,B 0,C 180,E1 -28251.007,E2 -28251.007} C_VEL
LIN {X 0,Y 61.995,Z 379.114,A -85,B 0,C 180,E1 -28260.001,E2 -28260.001} C_VEL
LIN {X 0,Y 58.477,Z 373.837,A -85,B 0,C 180,E1 -28269.951,E2 -28269.951} C_VEL
LIN {X 0,Y 56.792,Z 366.679,A -85,B 0,C 180,E1 -28281.795,E2 -28281.795} C_VEL
LIN {X 0,Y 56.855,Z 359.436,A -85,B 0,C 180,E1 -28291.69,E2 -28291.69} C_VEL
LIN {X 0,Y 57.53,Z 352.78,A -85,B 0,C 180,E1 -28299.119,E2 -28299.119} C_VEL
LIN {X 0,Y 57.633,Z 349.964,A -85,B 0,C 180,E1 -28301.844,E2 -28301.844} C_VEL
LIN {X 0,Y 57.036,Z 345.495,A -85,B 0,C 180,E1 -28305.697,E2 -28305.697} C_VEL
LIN {X 0,Y 55.006,Z 334.351,A -85,B 0,C 180,E1 -28314.148,E2 -28314.148} C_VEL
LIN {X 0,Y 55.191,Z 329.317,A -85,B 0,C 180,E1 -28317.482,E2 -28317.482} C_VEL
LIN {X 0,Y 55.544,Z 327.619,A -85,B 0,C 180,E1 -28318.492,E2 -28318.492} C_VEL
LIN {X 0,Y 58.785,Z 314.986,A -85,B 0,C 180,E1 -28324.71,E2 -28324.71} C_VEL
LIN {X 0,Y 61.648,Z 302.18,A -85,B 0,C 180,E1 -28329.085,E2 -28329.085} C_VEL
LIN {X 0,Y 63.865,Z 289.092,A -85,B 0,C 180,E1 -28332.146,E2 -28332.146} C_VEL
LIN {X 0,Y 67.27,Z 261.448,A -85,B 0,C 180,E1 -28336.14,E2 -28336.14} C_VEL
LIN {X 0,Y 69.752,Z 240.949,A -85,B 0,C 180,E1 -28338.771,E2 -28338.771} C_VEL
LIN {X 0,Y 63.981,Z 223.397,A -85,B 0,C 180,E1 -28344.873,E2 -28344.873} C_VEL
LIN {X 0,Y 59.515,Z 211.585,A -85,B 0,C 180,E1 -28350.1,E2 -28350.1} C_VEL
LIN {X 0,Y 56.371,Z 204.959,A -85,B 0,C 180,E1 -28354.111,E2 -28354.111} C_VEL
LIN {X 0,Y 54.146,Z 201.574,A -85,B 0,C 180,E1 -28357.044,E2 -28357.044} C_VEL
LIN {X 0,Y 52.174,Z 199.18,A -85,B 0,C 180,E1 -28359.809,E2 -28359.809} C_VEL
LIN {X 0,Y 51.509,Z 197.067,A -85,B 0,C 180,E1 -28361.304,E2 -28361.304} C_VEL
LIN {X 0,Y 51.336,Z 197.081,A -85,B 0,C 180,E1 -28366.594,E2 -28366.594} C_VEL
LIN {X 0,Y 50.995,Z 197.124,A -85,B 0,C 180,E1 -28374.414,E2 -28374.414} C_VEL
LIN {X 0,Y 50.983,Z 197.126,A -85,B 0,C 180,E1 -28384.194,E2 -28384.194} C_VEL
LIN {X 0,Y 50.973,Z 197.129,A -85,B 0,C 180,E1 -28393.572,E2 -28393.572} C_VEL
LIN {X 0,Y 51.006,Z 197.13,A -85,B 0,C 180,E1 -28405.752,E2 -28405.752} C_VEL
LIN {X 0,Y 50.993,Z 197.126,A -85,B 0,C 180,E1 -28415.575,E2 -28415.575} C_VEL
LIN {X 0,Y 51.387,Z 197.076,A -85,B 0,C 180,E1 -28424.123,E2 -28424.123} C_VEL
LIN {X 0,Y 51.641,Z 197.046,A -85,B 0,C 180,E1 -28432.176,E2 -28432.176} C_VEL
LIN {X 0,Y 52.21,Z 196.977,A -85,B 0,C 180,E1 -28439.998,E2 -28439.998} C_VEL
LIN {X 0,Y 51.631,Z 197.052,A -85,B 0,C 180,E1 -28447.822,E2 -28447.822} C_VEL
LIN {X 0,Y 51.394,Z 197.209,A -85,B 0,C 180,E1 -28456.125,E2 -28456.125} C_VEL
LIN {X 0,Y 52.254,Z 199.946,A -85,B 0,C 180,E1 -28457.893,E2 -28457.893} C_VEL
LIN {X 0,Y 53.869,Z 202.391,A -85,B 0,C 180,E1 -28460.275,E2 -28460.275} C_VEL
LIN {X 0,Y 57.768,Z 209.311,A -85,B 0,C 180,E1 -28465.441,E2 -28465.441} C_VEL
LIN {X 0,Y 62.181,Z 218.954,A -85,B 0,C 180,E1 -28470.57,E2 -28470.57} C_VEL
LIN {X 0,Y 66.032,Z 229.871,A -85,B 0,C 180,E1 -28474.894,E2 -28474.894} C_VEL
LIN {X 0,Y 69.457,Z 245.223,A -85,B 0,C 180,E1 -28479.226,E2 -28479.226} C_VEL
LIN {X 0,Y 69.15,Z 250.372,A -85,B 0,C 180,E1 -28480.005,E2 -28480.005} C_VEL
LIN {X 0,Y 64.265,Z 291.723,A -85,B 0,C 180,E1 -28485.808,E2 -28485.808} C_VEL
LIN {X 0,Y 61.732,Z 305.995,A -85,B 0,C 180,E1 -28489.117,E2 -28489.117} C_VEL
LIN {X 0,Y 59.012,Z 318.415,A -85,B 0,C 180,E1 -28493.461,E2 -28493.461} C_VEL
LIN {X 0,Y 55.812,Z 331.081,A -85,B 0,C 180,E1 -28499.763,E2 -28499.763} C_VEL
LIN {X 0,Y 53.413,Z 341.25,A -85,B 0,C 180,E1 -28506.758,E2 -28506.758} C_VEL
LIN {X 0,Y 51.79,Z 349.621,A -85,B 0,C 180,E1 -28514.259,E2 -28514.259} C_VEL
LIN {X 0,Y 50.998,Z 358.353,A -85,B 0,C 180,E1 -28524.074,E2 -28524.074} C_VEL
LIN {X 0,Y 51.359,Z 365.522,A -85,B 0,C 180,E1 -28533.93,E2 -28533.93} C_VEL
LIN {X 0,Y 51.67,Z 369.036,A -85,B 0,C 180,E1 -28539.796,E2 -28539.796} C_VEL
LIN {X 0,Y 53.261,Z 375.602,A -85,B 0,C 180,E1 -28553.327,E2 -28553.327} C_VEL
LIN {X 0,Y 58.418,Z 381.439,A -85,B 0,C 180,E1 -28566.986,E2 -28566.986} C_VEL
LIN {X 0,Y 66.518,Z 385.885,A -85,B 0,C 180,E1 -28577.704,E2 -28577.704} C_VEL
LIN {X 0,Y 76.718,Z 389.015,A -85,B 0,C 180,E1 -28585.542,E2 -28585.542} C_VEL
LIN {X 0,Y 82.356,Z 390.124,A -85,B 0,C 180,E1 -28588.588,E2 -28588.588} C_VEL
LIN {X 0,Y 84.814,Z 390.471,A -85,B 0,C 180,E1 -28590.187,E2 -28590.187} C_VEL
LIN {X 0,Y 72.547,Z 387.27,A -85,B 0,C 180,E1 -28597.202,E2 -28597.202} C_VEL
LIN {X 0,Y 64.48,Z 383.816,A -85,B 0,C 180,E1 -28604.25,E2 -28604.25} C_VEL
LIN {X 0,Y 57.897,Z 379.442,A -85,B 0,C 180,E1 -28613.029,E2 -28613.029} C_VEL
LIN {X 0,Y 52.488,Z 373.015,A -85,B 0,C 180,E1 -28625.765,E2 -28625.765} C_VEL
LIN {X 0,Y 50.204,Z 366.099,A -85,B 0,C 180,E1 -28638.361,E2 -28638.361} C_VEL
LIN {X 0,Y 49.902,Z 359.305,A -85,B 0,C 180,E1 -28648.816,E2 -28648.816} C_VEL
LIN {X 0,Y 50.581,Z 351.435,A -85,B 0,C 180,E1 -28658.719,E2 -28658.719} C_VEL
LIN {X 0,Y 52.257,Z 341.566,A -85,B 0,C 180,E1 -28668.465,E2 -28668.465} C_VEL
LIN {X 0,Y 54.772,Z 330.8,A -85,B 0,C 180,E1 -28676.519,E2 -28676.519} C_VEL
LIN {X 0,Y 55.544,Z 327.619,A -85,B 0,C 180,E1 -28678.492,E2 -28678.492} C_VEL
LIN {X 0,Y 56.196,Z 322.577,A -85,B 0,C 180,E1 -28681.35,E2 -28681.35} C_VEL
LIN {X 0,Y 55.573,Z 313.834,A -85,B 0,C 180,E1 -28685.971,E2 -28685.971} C_VEL
LIN {X 0,Y 54.913,Z 304.616,A -85,B 0,C 180,E1 -28690.171,E2 -28690.171} C_VEL
LIN {X 0,Y 55.504,Z 298.912,A -85,B 0,C 180,E1 -28692.119,E2 -28692.119} C_VEL
LIN {X 0,Y 57.685,Z 285.809,A -85,B 0,C 180,E1 -28695.14,E2 -28695.14} C_VEL
LIN {X 0,Y 60.969,Z 260.442,A -85,B 0,C 180,E1 -28698.989,E2 -28698.989} C_VEL
LIN {X 0,Y 63.311,Z 242.294,A -85,B 0,C 180,E1 -28701.465,E2 -28701.465} C_VEL
LIN {X 0,Y 57.963,Z 225.443,A -85,B 0,C 180,E1 -28708.049,E2 -28708.049} C_VEL
LIN {X 0,Y 54.324,Z 215.317,A -85,B 0,C 180,E1 -28713.242,E2 -28713.242} C_VEL
LIN {X 0,Y 51.817,Z 209.672,A -85,B 0,C 180,E1 -28717.139,E2 -28717.139} C_VEL
LIN {X 0,Y 50.137,Z 207.042,A -85,B 0,C 180,E1 -28719.741,E2 -28719.741} C_VEL
LIN {X 0,Y 47.803,Z 203.641,A -85,B 0,C 180,E1 -28723.694,E2 -28723.694} C_VEL
LIN {X 0,Y 47.032,Z 202.688,A -85,B 0,C 180,E1 -28725.069,E2 -28725.069} C_VEL
LIN {X 0,Y 44.687,Z 200.192,A -85,B 0,C 180,E1 -28729.672,E2 -28729.672} C_VEL
LIN {X 0,Y 43.969,Z 198.006,A -85,B 0,C 180,E1 -28732.035,E2 -28732.035} C_VEL
LIN {X 0,Y 43.81,Z 198.028,A -85,B 0,C 180,E1 -28738.759,E2 -28738.759} C_VEL
LIN {X 0,Y 43.781,Z 198.025,A -85,B 0,C 180,E1 -28749.938,E2 -28749.938} C_VEL
LIN {X 0,Y 43.824,Z 198.024,A -85,B 0,C 180,E1 -28763.293,E2 -28763.293} C_VEL
LIN {X 0,Y 43.808,Z 198.024,A -85,B 0,C 180,E1 -28771.228,E2 -28771.228} C_VEL
LIN {X 0,Y 44.174,Z 197.979,A -85,B 0,C 180,E1 -28782.639,E2 -28782.639} C_VEL
LIN {X 0,Y 44.487,Z 197.941,A -85,B 0,C 180,E1 -28790.908,E2 -28790.908} C_VEL
LIN {X 0,Y 45.085,Z 197.864,A -85,B 0,C 180,E1 -28799.998,E2 -28799.998} C_VEL
LIN {X 0,Y 44.625,Z 197.927,A -85,B 0,C 180,E1 -28806.498,E2 -28806.498} C_VEL
LIN {X 0,Y 45.562,Z 200.95,A -85,B 0,C 180,E1 -28809.418,E2 -28809.418} C_VEL
LIN {X 0,Y 47.38,Z 203.216,A -85,B 0,C 180,E1 -28812.951,E2 -28812.951} C_VEL
LIN {X 0,Y 52.647,Z 212.996,A -85,B 0,C 180,E1 -28822.002,E2 -28822.002} C_VEL
LIN {X 0,Y 56.545,Z 221.968,A -85,B 0,C 180,E1 -28827.528,E2 -28827.528} C_VEL
LIN {X 0,Y 60.148,Z 232.519,A -85,B 0,C 180,E1 -28832.214,E2 -28832.214} C_VEL
LIN {X 0,Y 63.119,Z 246.394,A -85,B 0,C 180,E1 -28836.65,E2 -28836.65} C_VEL
LIN {X 0,Y 60.744,Z 266.304,A -85,B 0,C 180,E1 -28839.487,E2 -28839.487} C_VEL
LIN {X 0,Y 57.56,Z 291.883,A -85,B 0,C 180,E1 -28843.543,E2 -28843.543} C_VEL
LIN {X 0,Y 54.892,Z 305.949,A -85,B 0,C 180,E1 -28847.151,E2 -28847.151} C_VEL
LIN {X 0,Y 51.774,Z 319.039,A -85,B 0,C 180,E1 -28852.358,E2 -28852.358} C_VEL
LIN {X 0,Y 48.55,Z 331.473,A -85,B 0,C 180,E1 -28859.572,E2 -28859.572} C_VEL
LIN {X 0,Y 46.019,Z 341.907,A -85,B 0,C 180,E1 -28868.119,E2 -28868.119} C_VEL
LIN {X 0,Y 44.415,Z 351.52,A -85,B 0,C 180,E1 -28878.6,E2 -28878.6} C_VEL
LIN {X 0,Y 44.241,Z 359.828,A -85,B 0,C 180,E1 -28890.008,E2 -28890.008} C_VEL
LIN {X 0,Y 44.97,Z 365.366,A -85,B 0,C 180,E1 -28898.999,E2 -28898.999} C_VEL
LIN {X 0,Y 45.611,Z 369.658,A -85,B 0,C 180,E1 -28907.957,E2 -28907.957} C_VEL
LIN {X 0,Y 49.674,Z 376.732,A -85,B 0,C 180,E1 -28924.475,E2 -28924.475} C_VEL
LIN {X 0,Y 55.089,Z 380.956,A -85,B 0,C 180,E1 -28934.569,E2 -28934.569} C_VEL
LIN {X 0,Y 62.065,Z 384.402,A -85,B 0,C 180,E1 -28942.443,E2 -28942.443} C_VEL
LIN {X 0,Y 67.346,Z 386.304,A -85,B 0,C 180,E1 -28946.61,E2 -28946.61} C_VEL
LIN {X 0,Y 71.627,Z 387.512,A -85,B 0,C 180,E1 -28950.621,E2 -28950.621} C_VEL
LIN {X 0,Y 60.209,Z 382.9,A -85,B 0,C 180,E1 -28959.052,E2 -28959.052} C_VEL
LIN {X 0,Y 52.546,Z 378.086,A -85,B 0,C 180,E1 -28968.428,E2 -28968.428} C_VEL
LIN {X 0,Y 46.34,Z 371.264,A -85,B 0,C 180,E1 -28982.175,E2 -28982.175} C_VEL
LIN {X 0,Y 43.719,Z 364.602,A -85,B 0,C 180,E1 -28995.277,E2 -28995.277} C_VEL
LIN {X 0,Y 43.12,Z 358.108,A -85,B 0,C 180,E1 -29006.632,E2 -29006.632} C_VEL
LIN {X 0,Y 43.696,Z 349.719,A -85,B 0,C 180,E1 -29018.528,E2 -29018.528} C_VEL
LIN {X 0,Y 45.624,Z 338.816,A -85,B 0,C 180,E1 -29030.376,E2 -29030.376} C_VEL
LIN {X 0,Y 48.271,Z 328.027,A -85,B 0,C 180,E1 -29038.967,E2 -29038.967} C_VEL
LIN {X 0,Y 51.819,Z 314.899,A -85,B 0,C 180,E1 -29046.312,E2 -29046.312} C_VEL
LIN {X 0,Y 54.789,Z 302.35,A -85,B 0,C 180,E1 -29051.095,E2 -29051.095} C_VEL
LIN {X 0,Y 55.504,Z 298.912,A -85,B 0,C 180,E1 -29052.119,E2 -29052.119} C_VEL
LIN {X 0,Y 55.983,Z 293.254,A -85,B 0,C 180,E1 -29053.803,E2 -29053.803} C_VEL
LIN {X 0,Y 53.328,Z 274.34,A -85,B 0,C 180,E1 -29059.66,E2 -29059.66} C_VEL
LIN {X 0,Y 53.609,Z 268.522,A -85,B 0,C 180,E1 -29060.826,E2 -29060.826} C_VEL
LIN {X 0,Y 56.865,Z 243.423,A -85,B 0,C 180,E1 -29064.678,E2 -29064.678} C_VEL
LIN {X 0,Y 52.329,Z 228.192,A -85,B 0,C 180,E1 -29071.603,E2 -29071.603} C_VEL
LIN {X 0,Y 49.273,Z 218.901,A -85,B 0,C 180,E1 -29077.134,E2 -29077.134} C_VEL
LIN {X 0,Y 47.306,Z 214.203,A -85,B 0,C 180,E1 -29080.798,E2 -29080.798} C_VEL
LIN {X 0,Y 43.638,Z 208.532,A -85,B 0,C 180,E1 -29088.07,E2 -29088.07} C_VEL
LIN {X 0,Y 41.343,Z 205.591,A -85,B 0,C 180,E1 -29093.823,E2 -29093.823} C_VEL
LIN {X 0,Y 40.776,Z 204.411,A -85,B 0,C 180,E1 -29095.743,E2 -29095.743} C_VEL
LIN {X 0,Y 38.072,Z 202.269,A -85,B 0,C 180,E1 -29104.97,E2 -29104.97} C_VEL
LIN {X 0,Y 36.593,Z 198.927,A -85,B 0,C 180,E1 -29115.913,E2 -29115.913} C_VEL
LIN {X 0,Y 36.702,Z 198.913,A -85,B 0,C 180,E1 -29124.934,E2 -29124.934} C_VEL
LIN {X 0,Y 37.12,Z 198.857,A -85,B 0,C 180,E1 -29142.751,E2 -29142.751} C_VEL
LIN {X 0,Y 37.172,Z 199.035,A -85,B 0,C 180,E1 -29145.66,E2 -29145.66} C_VEL
LIN {X 0,Y 38.818,Z 202.048,A -85,B 0,C 180,E1 -29154.804,E2 -29154.804} C_VEL
LIN {X 0,Y 41.211,Z 204.01,A -85,B 0,C 180,E1 -29162.444,E2 -29162.444} C_VEL
LIN {X 0,Y 42.6,Z 207.239,A -85,B 0,C 180,E1 -29166.87,E2 -29166.87} C_VEL
LIN {X 0,Y 43.69,Z 208.894,A -85,B 0,C 180,E1 -29169.502,E2 -29169.502} C_VEL
LIN {X 0,Y 48.125,Z 217.589,A -85,B 0,C 180,E1 -29178.602,E2 -29178.602} C_VEL
LIN {X 0,Y 51.482,Z 226.116,A -85,B 0,C 180,E1 -29184.499,E2 -29184.499} C_VEL
LIN {X 0,Y 54.408,Z 235.502,A -85,B 0,C 180,E1 -29189.236,E2 -29189.236} C_VEL
LIN {X 0,Y 56.849,Z 247.463,A -85,B 0,C 180,E1 -29193.568,E2 -29193.568} C_VEL
LIN {X 0,Y 51.013,Z 291.355,A -85,B 0,C 180,E1 -29200.747,E2 -29200.747} C_VEL
LIN {X 0,Y 48.171,Z 305.428,A -85,B 0,C 180,E1 -29204.674,E2 -29204.674} C_VEL
LIN {X 0,Y 45.103,Z 317.726,A -85,B 0,C 180,E1 -29210.012,E2 -29210.012} C_VEL
LIN {X 0,Y 41.61,Z 330.474,A -85,B 0,C 180,E1 -29218.297,E2 -29218.297} C_VEL
LIN {X 0,Y 38.851,Z 341.522,A -85,B 0,C 180,E1 -29228.8,E2 -29228.8} C_VEL
LIN {X 0,Y 37.434,Z 351.565,A -85,B 0,C 180,E1 -29241.915,E2 -29241.915} C_VEL
LIN {X 0,Y 37.874,Z 359.703,A -85,B 0,C 180,E1 -29255.333,E2 -29255.333} C_VEL
LIN {X 0,Y 38.671,Z 363.764,A -85,B 0,C 180,E1 -29263.14,E2 -29263.14} C_VEL
LIN {X 0,Y 41.261,Z 371.105,A -85,B 0,C 180,E1 -29280.739,E2 -29280.739} C_VEL
LIN {X 0,Y 46.154,Z 376.189,A -85,B 0,C 180,E1 -29293.264,E2 -29293.264} C_VEL
LIN {X 0,Y 55.404,Z 381.649,A -85,B 0,C 180,E1 -29305.551,E2 -29305.551} C_VEL
LIN {X 0,Y 58.108,Z 382.798,A -85,B 0,C 180,E1 -29307.858,E2 -29307.858} C_VEL
LIN {X 0,Y 59.918,Z 383.501,A -85,B 0,C 180,E1 -29310.492,E2 -29310.492} C_VEL
LIN {X 0,Y 50.144,Z 378.285,A -85,B 0,C 180,E1 -29319.491,E2 -29319.491} C_VEL
LIN {X 0,Y 42.582,Z 372.013,A -85,B 0,C 180,E1 -29332.062,E2 -29332.062} C_VEL
LIN {X 0,Y 37.891,Z 364.523,A -85,B 0,C 180,E1 -29347.999,E2 -29347.999} C_VEL
LIN {X 0,Y 36.477,Z 357.248,A -85,B 0,C 180,E1 -29362.668,E2 -29362.668} C_VEL
LIN {X 0,Y 36.597,Z 349.891,A -85,B 0,C 180,E1 -29375.181,E2 -29375.181} C_VEL
LIN {X 0,Y 37.994,Z 340.619,A -85,B 0,C 180,E1 -29387.727,E2 -29387.727} C_VEL
LIN {X 0,Y 40.378,Z 331.004,A -85,B 0,C 180,E1 -29397.45,E2 -29397.45} C_VEL
LIN {X 0,Y 43.72,Z 318.951,A -85,B 0,C 180,E1 -29406.108,E2 -29406.108} C_VEL
LIN {X 0,Y 46.997,Z 306.579,A -85,B 0,C 180,E1 -29412.058,E2 -29412.058} C_VEL
LIN {X 0,Y 49.945,Z 293.235,A -85,B 0,C 180,E1 -29416.332,E2 -29416.332} C_VEL
LIN {X 0,Y 52.546,Z 276.151,A -85,B 0,C 180,E1 -29419.625,E2 -29419.625} C_VEL
LIN {X 0,Y 53.609,Z 268.522,A -85,B 0,C 180,E1 -29420.826,E2 -29420.826} C_VEL
LIN {X 0,Y 54.052,Z 262.688,A -85,B 0,C 180,E1 -29421.929,E2 -29421.929} C_VEL
LIN {X 0,Y 53.633,Z 256.931,A -85,B 0,C 180,E1 -29423.52,E2 -29423.52} C_VEL
LIN {X 0,Y 52.157,Z 249.463,A -85,B 0,C 180,E1 -29426.286,E2 -29426.286} C_VEL
LIN {X 0,Y 49.092,Z 238.659,A -85,B 0,C 180,E1 -29431.56,E2 -29431.56} C_VEL
LIN {X 0,Y 45.002,Z 224.235,A -85,B 0,C 180,E1 -29440.294,E2 -29440.294} C_VEL
LIN {X 0,Y 42.98,Z 218.726,A -85,B 0,C 180,E1 -29445.095,E2 -29445.095} C_VEL
LIN {X 0,Y 40.125,Z 214.105,A -85,B 0,C 180,E1 -29452.292,E2 -29452.292} C_VEL
LIN {X 0,Y 38.099,Z 210.785,A -85,B 0,C 180,E1 -29459.159,E2 -29459.159} C_VEL
LIN {X 0,Y 35.774,Z 208.392,A -85,B 0,C 180,E1 -29469.322,E2 -29469.322} C_VEL
LIN {X 0,Y 34.849,Z 205.767,A -85,B 0,C 180,E1 -29479.044,E2 -29479.044} C_VEL
LIN {X 0,Y 35.322,Z 205.869,A -85,B 0,C 180,E1 -29502.614,E2 -29502.614} C_VEL
LIN {X 0,Y 37.28,Z 209.149,A -85,B 0,C 180,E1 -29514.589,E2 -29514.589} C_VEL
LIN {X 0,Y 38.283,Z 210.16,A -85,B 0,C 180,E1 -29518.354,E2 -29518.354} C_VEL
LIN {X 0,Y 40.901,Z 215.936,A -85,B 0,C 180,E1 -29527.524,E2 -29527.524} C_VEL
LIN {X 0,Y 43.991,Z 222.918,A -85,B 0,C 180,E1 -29535.275,E2 -29535.275} C_VEL
LIN {X 0,Y 46.907,Z 231.282,A -85,B 0,C 180,E1 -29541.499,E2 -29541.499} C_VEL
LIN {X 0,Y 48.741,Z 237.898,A -85,B 0,C 180,E1 -29545.305,E2 -29545.305} C_VEL
LIN {X 0,Y 50.669,Z 248.454,A -85,B 0,C 180,E1 -29549.77,E2 -29549.77} C_VEL
LIN {X 0,Y 44.619,Z 290.762,A -85,B 0,C 180,E1 -29557.131,E2 -29557.131} C_VEL
LIN {X 0,Y 41.578,Z 304.926,A -85,B 0,C 180,E1 -29561.416,E2 -29561.416} C_VEL
LIN {X 0,Y 38.558,Z 316.31,A -85,B 0,C 180,E1 -29566.807,E2 -29566.807} C_VEL
LIN {X 0,Y 35.046,Z 328.026,A -85,B 0,C 180,E1 -29575.232,E2 -29575.232} C_VEL
LIN {X 0,Y 32.083,Z 339.248,A -85,B 0,C 180,E1 -29587.471,E2 -29587.471} C_VEL
LIN {X 0,Y 30.659,Z 349.579,A -85,B 0,C 180,E1 -29603.43,E2 -29603.43} C_VEL
LIN {X 0,Y 31.522,Z 357.981,A -85,B 0,C 180,E1 -29619.637,E2 -29619.637} C_VEL
LIN {X 0,Y 32.631,Z 362.104,A -85,B 0,C 180,E1 -29628.86,E2 -29628.86} C_VEL
LIN {X 0,Y 35.737,Z 368.599,A -85,B 0,C 180,E1 -29646.167,E2 -29646.167} C_VEL
LIN {X 0,Y 43.855,Z 375.54,A -85,B 0,C 180,E1 -29663.264,E2 -29663.264} C_VEL
LIN {X 0,Y 49.041,Z 378.47,A -85,B 0,C 180,E1 -29669.312,E2 -29669.312} C_VEL
LIN {X 0,Y 48.476,Z 378.135,A -85,B 0,C 180,E1 -29670.458,E2 -29670.458} C_VEL
LIN {X 0,Y 38.272,Z 370.83,A -85,B 0,C 180,E1 -29684.013,E2 -29684.013} C_VEL
LIN {X 0,Y 31.804,Z 362.304,A -85,B 0,C 180,E1 -29703.17,E2 -29703.17} C_VEL
LIN {X 0,Y 29.904,Z 355.045,A -85,B 0,C 180,E1 -29719.905,E2 -29719.905} C_VEL
LIN {X 0,Y 29.901,Z 346.868,A -85,B 0,C 180,E1 -29735.992,E2 -29735.992} C_VEL
LIN {X 0,Y 31.65,Z 336.519,A -85,B 0,C 180,E1 -29751.631,E2 -29751.631} C_VEL
LIN {X 0,Y 34.3,Z 326.81,A -85,B 0,C 180,E1 -29762.178,E2 -29762.178} C_VEL
LIN {X 0,Y 38.056,Z 314.593,A -85,B 0,C 180,E1 -29771.173,E2 -29771.173} C_VEL
LIN {X 0,Y 41.47,Z 302.083,A -85,B 0,C 180,E1 -29777.033,E2 -29777.033} C_VEL
LIN {X 0,Y 44.009,Z 289.855,A -85,B 0,C 180,E1 -29780.803,E2 -29780.803} C_VEL
LIN {X 0,Y 48.319,Z 261.816,A -85,B 0,C 180,E1 -29785.827,E2 -29785.827} C_VEL
LIN {X 0,Y 50.753,Z 245.035,A -85,B 0,C 180,E1 -29788.44,E2 -29788.44} C_VEL
LIN {X 0,Y 49.092,Z 238.659,A -85,B 0,C 180,E1 -29791.56,E2 -29791.56} C_VEL
LIN {X 0,Y 47.125,Z 233.79,A -85,B 0,C 180,E1 -29794.882,E2 -29794.882} C_VEL
LIN {X 0,Y 43.651,Z 228.315,A -85,B 0,C 180,E1 -29800.733,E2 -29800.733} C_VEL
LIN {X 0,Y 39.095,Z 222.592,A -85,B 0,C 180,E1 -29810.52,E2 -29810.52} C_VEL
LIN {X 0,Y 36.127,Z 218.364,A -85,B 0,C 180,E1 -29820.189,E2 -29820.189} C_VEL
LIN {X 0,Y 35.332,Z 216.957,A -85,B 0,C 180,E1 -29823.836,E2 -29823.836} C_VEL
LIN {X 0,Y 33.632,Z 214.194,A -85,B 0,C 180,E1 -29835.276,E2 -29835.276} C_VEL
LIN {X 0,Y 33.361,Z 212.761,A -85,B 0,C 180,E1 -29840.799,E2 -29840.799} C_VEL
LIN {X 0,Y 33.662,Z 212.788,A -85,B 0,C 180,E1 -29860.15,E2 -29860.15} C_VEL
LIN {X 0,Y 35.633,Z 216.451,A -85,B 0,C 180,E1 -29874.169,E2 -29874.169} C_VEL
LIN {X 0,Y 37.614,Z 221.511,A -85,B 0,C 180,E1 -29883.182,E2 -29883.182} C_VEL
LIN {X 0,Y 39.965,Z 228.053,A -85,B 0,C 180,E1 -29891.142,E2 -29891.142} C_VEL
LIN {X 0,Y 42.188,Z 235.927,A -85,B 0,C 180,E1 -29897.565,E2 -29897.565} C_VEL
LIN {X 0,Y 43.529,Z 241.633,A -85,B 0,C 180,E1 -29901.153,E2 -29901.153} C_VEL
LIN {X 0,Y 44.724,Z 249.415,A -85,B 0,C 180,E1 -29904.89,E2 -29904.89} C_VEL
LIN {X 0,Y 38.459,Z 290.055,A -85,B 0,C 180,E1 -29912.388,E2 -29912.388} C_VEL
LIN {X 0,Y 35.181,Z 304.125,A -85,B 0,C 180,E1 -29916.976,E2 -29916.976} C_VEL
LIN {X 0,Y 31.56,Z 316.481,A -85,B 0,C 180,E1 -29923.648,E2 -29923.648} C_VEL
LIN {X 0,Y 27.554,Z 329.067,A -85,B 0,C 180,E1 -29935.013,E2 -29935.013} C_VEL
LIN {X 0,Y 24.661,Z 340.289,A -85,B 0,C 180,E1 -29951.315,E2 -29951.315} C_VEL
LIN {X 0,Y 24.227,Z 351.189,A -85,B 0,C 180,E1 -29974.173,E2 -29974.173} C_VEL
LIN {X 0,Y 25.952,Z 357.687,A -85,B 0,C 180,E1 -29989.8,E2 -29989.8} C_VEL
LIN {X 0,Y 27.576,Z 361.509,A -85,B 0,C 180,E1 -30000.66,E2 -30000.66} C_VEL
LIN {X 0,Y 34.165,Z 369.114,A -85,B 0,C 180,E1 -30021.896,E2 -30021.896} C_VEL
LIN {X 0,Y 38.535,Z 372.242,A -85,B 0,C 180,E1 -30029.277,E2 -30029.277} C_VEL
LIN {X 0,Y 30.102,Z 365.14,A -85,B 0,C 180,E1 -30043.214,E2 -30043.214} C_VEL
LIN {X 0,Y 24.735,Z 356.942,A -85,B 0,C 180,E1 -30064.077,E2 -30064.077} C_VEL
LIN {X 0,Y 23.079,Z 349.373,A -85,B 0,C 180,E1 -30083.962,E2 -30083.962} C_VEL
LIN {X 0,Y 23.497,Z 341.103,A -85,B 0,C 180,E1 -30102.303,E2 -30102.303} C_VEL
LIN {X 0,Y 26.162,Z 330.133,A -85,B 0,C 180,E1 -30120.038,E2 -30120.038} C_VEL
LIN {X 0,Y 30.137,Z 317.693,A -85,B 0,C 180,E1 -30132.511,E2 -30132.511} C_VEL
LIN {X 0,Y 33.974,Z 305.412,A -85,B 0,C 180,E1 -30139.914,E2 -30139.914} C_VEL
LIN {X 0,Y 37.273,Z 292.246,A -85,B 0,C 180,E1 -30144.787,E2 -30144.787} C_VEL
LIN {X 0,Y 40.967,Z 271.024,A -85,B 0,C 180,E1 -30149.169,E2 -30149.169} C_VEL
LIN {X 0,Y 44.852,Z 246.505,A -85,B 0,C 180,E1 -30153.24,E2 -30153.24} C_VEL
LIN {X 0,Y 41.637,Z 233.193,A -85,B 0,C 180,E1 -30161.542,E2 -30161.542} C_VEL
LIN {X 0,Y 39.758,Z 225.755,A -85,B 0,C 180,E1 -30167.613,E2 -30167.613} C_VEL
LIN {X 0,Y 38.847,Z 223.143,A -85,B 0,C 180,E1 -30170.602,E2 -30170.602} C_VEL
LIN {X 0,Y 36.845,Z 219.514,A -85,B 0,C 180,E1 -30177.404,E2 -30177.404} C_VEL
LIN {X 0,Y 36.127,Z 218.364,A -85,B 0,C 180,E1 -30180.189,E2 -30180.189} C_VEL
LIN {X 0,Y 35.04,Z 217.251,A -85,B 0,C 180,E1 -30184.72,E2 -30184.72} C_VEL
LIN {X 0,Y 33.54,Z 217.158,A -85,B 0,C 180,E1 -30191.975,E2 -30191.975} C_VEL
LIN {X 0,Y 31.863,Z 219.577,A -85,B 0,C 180,E1 -30213.411,E2 -30213.411} C_VEL
LIN {X 0,Y 31.976,Z 219.644,A -85,B 0,C 180,E1 -30215.917,E2 -30215.917} C_VEL
LIN {X 0,Y 32.194,Z 220.219,A -85,B 0,C 180,E1 -30219.897,E2 -30219.897} C_VEL
LIN {X 0,Y 33.198,Z 222.686,A -85,B 0,C 180,E1 -30229.515,E2 -30229.515} C_VEL
LIN {X 0,Y 34.378,Z 226.639,A -85,B 0,C 180,E1 -30237.202,E2 -30237.202} C_VEL
LIN {X 0,Y 36.028,Z 232.59,A -85,B 0,C 180,E1 -30245.437,E2 -30245.437} C_VEL
LIN {X 0,Y 38.179,Z 242.551,A -85,B 0,C 180,E1 -30254.354,E2 -30254.354} C_VEL
LIN {X 0,Y 39.098,Z 250.463,A -85,B 0,C 180,E1 -30258.884,E2 -30258.884} C_VEL
LIN {X 0,Y 32.522,Z 289.455,A -85,B 0,C 180,E1 -30266.149,E2 -30266.149} C_VEL
LIN {X 0,Y 29.071,Z 303.194,A -85,B 0,C 180,E1 -30270.752,E2 -30270.752} C_VEL
LIN {X 0,Y 24.772,Z 316.497,A -85,B 0,C 180,E1 -30278.744,E2 -30278.744} C_VEL
LIN {X 0,Y 20.348,Z 328.96,A -85,B 0,C 180,E1 -30292.834,E2 -30292.834} C_VEL
LIN {X 0,Y 17.531,Z 340.145,A -85,B 0,C 180,E1 -30315.51,E2 -30315.51} C_VEL
LIN {X 0,Y 18.483,Z 350.855,A -85,B 0,C 180,E1 -30346.589,E2 -30346.589} C_VEL
LIN {X 0,Y 20.709,Z 355.701,A -85,B 0,C 180,E1 -30360.621,E2 -30360.621} C_VEL
LIN {X 0,Y 23.19,Z 359.597,A -85,B 0,C 180,E1 -30373.01,E2 -30373.01} C_VEL
LIN {X 0,Y 26.357,Z 363.026,A -85,B 0,C 180,E1 -30383.146,E2 -30383.146} C_VEL
LIN {X 0,Y 27.678,Z 364.219,A -85,B 0,C 180,E1 -30389.484,E2 -30389.484} C_VEL
LIN {X 0,Y 20.092,Z 355.829,A -85,B 0,C 180,E1 -30409.922,E2 -30409.922} C_VEL
LIN {X 0,Y 16.826,Z 347.905,A -85,B 0,C 180,E1 -30435.138,E2 -30435.138} C_VEL
LIN {X 0,Y 16.732,Z 338.657,A -85,B 0,C 180,E1 -30463.039,E2 -30463.039} C_VEL
LIN {X 0,Y 20.081,Z 326.776,A -85,B 0,C 180,E1 -30487.177,E2 -30487.177} C_VEL
LIN {X 0,Y 24.506,Z 314.553,A -85,B 0,C 180,E1 -30500.369,E2 -30500.369} C_VEL
LIN {X 0,Y 28.654,Z 301.977,A -85,B 0,C 180,E1 -30507.64,E2 -30507.64} C_VEL
LIN {X 0,Y 31.818,Z 289.519,A -85,B 0,C 180,E1 -30511.927,E2 -30511.927} C_VEL
LIN {X 0,Y 37.096,Z 259.92,A -85,B 0,C 180,E1 -30517.496,E2 -30517.496} C_VEL
LIN {X 0,Y 39.138,Z 247.163,A -85,B 0,C 180,E1 -30519.693,E2 -30519.693} C_VEL
LIN {X 0,Y 36.498,Z 233.463,A -85,B 0,C 180,E1 -30530.448,E2 -30530.448} C_VEL
LIN {X 0,Y 35.455,Z 228.37,A -85,B 0,C 180,E1 -30535.881,E2 -30535.881} C_VEL
LIN {X 0,Y 33.759,Z 224.774,A -85,B 0,C 180,E1 -30543.614,E2 -30543.614} C_VEL
LIN {X 0,Y 33.074,Z 223.333,A -85,B 0,C 180,E1 -30547.789,E2 -30547.789} C_VEL
LIN {X 0,Y 31.873,Z 219.693,A -85,B 0,C 180,E1 -30563.718,E2 -30563.718} C_VEL
LIN {X 0,Y 31.976,Z 219.644,A -85,B 0,C 180,E1 -30575.917,E2 -30575.917} C_VEL
LIN {X 0,Y 32.204,Z 220.29,A -85,B 0,C 180,E1 -30580.12,E2 -30580.12} C_VEL
LIN {X 0,Y 32.403,Z 222.747,A -85,B 0,C 180,E1 -30585.274,E2 -30585.274} C_VEL
LIN {X 0,Y 32.417,Z 226.077,A -85,B 0,C 180,E1 -30589.061,E2 -30589.061} C_VEL
LIN {X 0,Y 32.294,Z 235.665,A -85,B 0,C 180,E1 -30596.788,E2 -30596.788} C_VEL
LIN {X 0,Y 32.412,Z 236.958,A -85,B 0,C 180,E1 -30598.123,E2 -30598.123} C_VEL
LIN {X 0,Y 33.613,Z 245.45,A -85,B 0,C 180,E1 -30606.862,E2 -30606.862} C_VEL
LIN {X 0,Y 34.021,Z 251.229,A -85,B 0,C 180,E1 -30610.858,E2 -30610.858} C_VEL
LIN {X 0,Y 27.235,Z 288.446,A -85,B 0,C 180,E1 -30617.25,E2 -30617.25} C_VEL
LIN {X 0,Y 23.74,Z 301.47,A -85,B 0,C 180,E1 -30621.079,E2 -30621.079} C_VEL
LIN {X 0,Y 19.027,Z 314.64,A -85,B 0,C 180,E1 -30628.726,E2 -30628.726} C_VEL
LIN {X 0,Y 14.362,Z 325.947,A -85,B 0,C 180,E1 -30642.81,E2 -30642.81} C_VEL
LIN {X 0,Y 10.844,Z 337.472,A -85,B 0,C 180,E1 -30675.967,E2 -30675.967} C_VEL
LIN {X 0,Y 12.274,Z 346.802,A -85,B 0,C 180,E1 -30715.463,E2 -30715.463} C_VEL
LIN {X 0,Y 16.67,Z 353.662,A -85,B 0,C 180,E1 -30737.574,E2 -30737.574} C_VEL
LIN {X 0,Y 17.845,Z 355.062,A -85,B 0,C 180,E1 -30742,E2 -30742} C_VEL
LIN {X 0,Y 17.524,Z 354.836,A -85,B 0,C 180,E1 -30748.766,E2 -30748.766} C_VEL
LIN {X 0,Y 12.096,Z 347.681,A -85,B 0,C 180,E1 -30771.647,E2 -30771.647} C_VEL
LIN {X 0,Y 9.751,Z 339.517,A -85,B 0,C 180,E1 -30808.686,E2 -30808.686} C_VEL
LIN {X 0,Y 12.26,Z 328.62,A -85,B 0,C 180,E1 -30848.666,E2 -30848.666} C_VEL
LIN {X 0,Y 17.66,Z 315.709,A -85,B 0,C 180,E1 -30868.561,E2 -30868.561} C_VEL
LIN {X 0,Y 22.556,Z 302.892,A -85,B 0,C 180,E1 -30876.669,E2 -30876.669} C_VEL
LIN {X 0,Y 26.273,Z 290.19,A -85,B 0,C 180,E1 -30880.805,E2 -30880.805} C_VEL
LIN {X 0,Y 32.08,Z 260.307,A -85,B 0,C 180,E1 -30885.859,E2 -30885.859} C_VEL
LIN {X 0,Y 34.159,Z 248.824,A -85,B 0,C 180,E1 -30887.512,E2 -30887.512} C_VEL
LIN {X 0,Y 32.461,Z 235.136,A -85,B 0,C 180,E1 -30900.322,E2 -30900.322} C_VEL
LIN {X 0,Y 31.99,Z 232.743,A -85,B 0,C 180,E1 -30903.98,E2 -30903.98} C_VEL
LIN {X 0,Y 31.032,Z 229.723,A -85,B 0,C 180,E1 -30911.991,E2 -30911.991} C_VEL
LIN {X 0,Y 30.483,Z 226.605,A -85,B 0,C 180,E1 -30926.559,E2 -30926.559} C_VEL
LIN {X 0,Y 30.594,Z 226.751,A -85,B 0,C 180,E1 -30935.605,E2 -30935.605} C_VEL
LIN {X 0,Y 31,Z 228.69,A -85,B 0,C 180,E1 -30943.747,E2 -30943.747} C_VEL
LIN {X 0,Y 31.702,Z 233.144,A -85,B 0,C 180,E1 -30952.479,E2 -30952.479} C_VEL
LIN {X 0,Y 32.412,Z 236.958,A -85,B 0,C 180,E1 -30958.123,E2 -30958.123} C_VEL
LIN {X 0,Y 32.57,Z 240.49,A -85,B 0,C 180,E1 -30961.003,E2 -30961.003} C_VEL
LIN {X 0,Y 32.013,Z 246.244,A -85,B 0,C 180,E1 -30963.111,E2 -30963.111} C_VEL
LIN {X 0,Y 30.773,Z 252.098,A -85,B 0,C 180,E1 -30963.435,E2 -30963.435} C_VEL
LIN {X 0,Y 27.517,Z 264.22,A -85,B 0,C 180,E1 -30962.088,E2 -30962.088} C_VEL
LIN {X 0,Y 26.632,Z 268.302,A -85,B 0,C 180,E1 -30962.275,E2 -30962.275} C_VEL
LIN {X 0,Y 21.828,Z 291.231,A -85,B 0,C 180,E1 -30965.231,E2 -30965.231} C_VEL
LIN {X 0,Y 17.733,Z 304.02,A -85,B 0,C 180,E1 -30967.914,E2 -30967.914} C_VEL
LIN {X 0,Y 12.652,Z 316.019,A -85,B 0,C 180,E1 -30973.681,E2 -30973.681} C_VEL
LIN {X 0,Y 6.428,Z 328.322,A -85,B 0,C 180,E1 -30995.005,E2 -30995.005} C_VEL
LIN {X 0,Y 5.039,Z 339.299,A -85,B 0,C 180,E1 -31081.613,E2 -31081.613} C_VEL
LIN {X 0,Y 5.589,Z 340.358,A -85,B 0,C 180,E1 -31089.039,E2 -31089.039} C_VEL
LIN {X 0,Y 6.617,Z 342.152,A -85,B 0,C 180,E1 -31107.94,E2 -31107.94} C_VEL
LIN {X 0,Y 3.492,Z 332.621,A -85,B 0,C 180,E1 -31197.442,E2 -31197.442} C_VEL
LIN {X 0,Y 8.952,Z 321.825,A -85,B 0,C 180,E1 -31241.025,E2 -31241.025} C_VEL
LIN {X 0,Y 14.919,Z 309.602,A -85,B 0,C 180,E1 -31249.561,E2 -31249.561} C_VEL
LIN {X 0,Y 19.928,Z 296.117,A -85,B 0,C 180,E1 -31252.939,E2 -31252.939} C_VEL
LIN {X 0,Y 23.391,Z 282.559,A -85,B 0,C 180,E1 -31254.847,E2 -31254.847} C_VEL
LIN {X 0,Y 29.895,Z 250.347,A -85,B 0,C 180,E1 -31257.718,E2 -31257.718} C_VEL
LIN {X 0,Y 29.465,Z 238.11,A -85,B 0,C 180,E1 -31271.229,E2 -31271.229} C_VEL
LIN {X 0,Y 29.11,Z 235.971,A -85,B 0,C 180,E1 -31277.735,E2 -31277.735} C_VEL
LIN {X 0,Y 29.094,Z 233.641,A -85,B 0,C 180,E1 -31289.16,E2 -31289.16} C_VEL
LIN {X 0,Y 29.132,Z 233.738,A -85,B 0,C 180,E1 -31293.097,E2 -31293.097} C_VEL
LIN {X 0,Y 29.152,Z 235.181,A -85,B 0,C 180,E1 -31298.467,E2 -31298.467} C_VEL
LIN {X 0,Y 29.323,Z 240.398,A -85,B 0,C 180,E1 -31308.11,E2 -31308.11} C_VEL
LIN {X 0,Y 29.738,Z 248.565,A -85,B 0,C 180,E1 -31317.673,E2 -31317.673} C_VEL
LIN {X 0,Y 29.637,Z 253.03,A -85,B 0,C 180,E1 -31320.69,E2 -31320.69} C_VEL
LIN {X 0,Y 26.632,Z 268.302,A -85,B 0,C 180,E1 -31322.275,E2 -31322.275} C_VEL
LIN {X 0,Y 25.196,Z 274.029,A -85,B 0,C 180,E1 -31321.794,E2 -31321.794} C_VEL
LIN {X 0,Y 21.899,Z 283.132,A -85,B 0,C 180,E1 -31316.467,E2 -31316.467} C_VEL
LIN {X 0,Y 18.525,Z 292.137,A -85,B 0,C 180,E1 -31308.748,E2 -31308.748} C_VEL
LIN {X 0,Y 16.612,Z 297.724,A -85,B 0,C 180,E1 -31306.191,E2 -31306.191} C_VEL
LIN {X 0,Y 11.925,Z 310.068,A -85,B 0,C 180,E1 -31303.174,E2 -31303.174} C_VEL
LIN {X 0,Y 7.659,Z 318.968,A -85,B 0,C 180,E1 -31296.463,E2 -31296.463} C_VEL
LIN {X 0,Y 8.558,Z 316.986,A -85,B 0,C 180,E1 -31285.134,E2 -31285.134} C_VEL
LIN {X 0,Y 13.342,Z 306.196,A -85,B 0,C 180,E1 -31276.251,E2 -31276.251} C_VEL
LIN {X 0,Y 17.923,Z 292.829,A -85,B 0,C 180,E1 -31272.665,E2 -31272.665} C_VEL
LIN {X 0,Y 22.574,Z 272.372,A -85,B 0,C 180,E1 -31271.065,E2 -31271.065} C_VEL
LIN {X 0,Y 26.806,Z 251.322,A -85,B 0,C 180,E1 -31271.262,E2 -31271.262} C_VEL
LIN {X 0,Y 27.514,Z 242.8,A -85,B 0,C 180,E1 -31281.557,E2 -31281.557} C_VEL
LIN {X 0,Y 27.637,Z 241.196,A -85,B 0,C 180,E1 -31289.425,E2 -31289.425} C_VEL
LIN {X 0,Y 27.618,Z 241.351,A -85,B 0,C 180,E1 -31291.146,E2 -31291.146} C_VEL
LIN {X 0,Y 27.131,Z 245.695,A -85,B 0,C 180,E1 -31298.878,E2 -31298.878} C_VEL
LIN {X 0,Y 26.674,Z 252.348,A -85,B 0,C 180,E1 -31306.665,E2 -31306.665} C_VEL
LIN {X 0,Y 26.419,Z 254.263,A -85,B 0,C 180,E1 -31307.568,E2 -31307.568} C_VEL
LIN {X 0,Y 19.131,Z 289.221,A -85,B 0,C 180,E1 -31307.293,E2 -31307.293} C_VEL
LIN {X 0,Y 16.612,Z 297.724,A -85,B 0,C 180,E1 -31306.191,E2 -31306.191} C_VEL
LIN {X 0,Y 16.712,Z 296.583,A -85,B 0,C 180,E1 -31302.833,E2 -31302.833} C_VEL
LIN {X 0,Y 17.992,Z 290.7,A -85,B 0,C 180,E1 -31297.089,E2 -31297.089} C_VEL
LIN {X 0,Y 22.268,Z 269.624,A -85,B 0,C 180,E1 -31286.954,E2 -31286.954} C_VEL
LIN {X 0,Y 24.258,Z 259.11,A -85,B 0,C 180,E1 -31285.52,E2 -31285.52} C_VEL
LIN {X 0,Y 25.421,Z 252.826,A -85,B 0,C 180,E1 -31286.848,E2 -31286.848} C_VEL
LIN {X 0,Y 25.654,Z 251.49,A -85,B 0,C 180,E1 -31288.695,E2 -31288.695} C_VEL
LIN {X 0,Y 25.146,Z 254.225,A -85,B 0,C 180,E1 -31291.872,E2 -31291.872} C_VEL
LIN {X 0,Y 23.629,Z 261.973,A -85,B 0,C 180,E1 -31290.934,E2 -31290.934} C_VEL
LIN {X 0,Y 23.632,Z 261.972,A -85,B 0,C 180,E1 -31287.779,E2 -31287.779} C_VEL
LIN {X 0,Y 25.421,Z 252.826,A -85,B 0,C 180,E1 -31286.848,E2 -31286.848} C_VEL
LIN {X 0,Y 28.501,Z 253.309,A -85,B 0,C 180,E1 -31292.082,E2 -31292.082} C_VEL
LIN {X 0,Y 28.501,Z 600,A -85,B 0,C 180,E1 -31292.082,E2 -31292.082} C_VEL
LIN {X 0,Y 28.501,Z 600,A -85,B 0,C 180,E1 -31292.082,E2 -31292.082}

QRS_NEXT_CUT()

QRS_NEXT()
QRS_HOME()

END
